	bArm2VertULD1Up_00 AT %MX26056.0 : BOOL;
	bArm2VertULD1Up_01 AT %MX26056.1 : BOOL;
	bArm2VertULD1Up_02 AT %MX26056.2 : BOOL;
	bArm2VertULD1Up_03 AT %MX26056.3 : BOOL;
	bArm2VertULD1Up_04 AT %MX26056.4 : BOOL;
	bArm2VertULD1Up_05 AT %MX26056.5 : BOOL;
	bArm2VertULD1Up_06 AT %MX26056.6 : BOOL;
	bArm2VertULD1Up_07 AT %MX26056.7 : BOOL;
	bArm2VertULD1Up_08 AT %MX26056.8 : BOOL;
	bArm2VertULD1Up_09 AT %MX26056.9 : BOOL;
	bArm2VertULD1Up_10 AT %MX26056.10 : BOOL;
	bArm2VertULD1Up_11 AT %MX26056.11 : BOOL;
	bArm2VertULD1Up_12 AT %MX26056.12 : BOOL;
	bArm2VertULD1Up_13 AT %MX26056.13 : BOOL;
	bArm2VertULD1Up_14 AT %MX26056.14 : BOOL;
	bArm2VertULD1Up_15 AT %MX26056.15 : BOOL;
	bArm2VertULD1Up_16 AT %MX26056.16 : BOOL;
	bArm2VertULD1Up_17 AT %MX26056.17 : BOOL;
	bArm2VertULD1Up_18 AT %MX26056.18 : BOOL;
	bArm2VertULD1Up_19 AT %MX26056.19 : BOOL;
	bArm2VertULD1Up_20 AT %MX26056.20 : BOOL;
	bArm2VertULD1Up_21 AT %MX26056.21 : BOOL;
	bArm2VertULD1Up_22 AT %MX26056.22 : BOOL;
	bArm2VertULD1Up_23 AT %MX26056.23 : BOOL;
	bArm2VertULD1Up_24 AT %MX26056.24 : BOOL;
	bArm2VertULD1Up_25 AT %MX26056.25 : BOOL;
	bArm2VertULD1Up_26 AT %MX26056.26 : BOOL;
	bArm2VertULD1Up_27 AT %MX26056.27 : BOOL;
	bArm2VertULD1Up_28 AT %MX26056.28 : BOOL;
	bArm2VertULD1Up_29 AT %MX26056.29 : BOOL;
	bArm2VertULD1Up_30 AT %MX26056.30 : BOOL;
	bArm2VertULD1Up_31 AT %MX26056.31 : BOOL;

	bArm2VertStn1Up_00 AT %MX26004.0 : BOOL;
	bArm2VertStn1Up_01 AT %MX26004.1 : BOOL;
	bArm2VertStn1Up_02 AT %MX26004.2 : BOOL;
	bArm2VertStn1Up_03 AT %MX26004.3 : BOOL;
	bArm2VertStn1Up_04 AT %MX26004.4 : BOOL;
	bArm2VertStn1Up_05 AT %MX26004.5 : BOOL;
	bArm2VertStn1Up_06 AT %MX26004.6 : BOOL;
	bArm2VertStn1Up_07 AT %MX26004.7 : BOOL;
	bArm2VertStn1Up_08 AT %MX26004.8 : BOOL;
	bArm2VertStn1Up_09 AT %MX26004.9 : BOOL;
	bArm2VertStn1Up_10 AT %MX26004.10 : BOOL;
	bArm2VertStn1Up_11 AT %MX26004.11 : BOOL;
	bArm2VertStn1Up_12 AT %MX26004.12 : BOOL;
	bArm2VertStn1Up_13 AT %MX26004.13 : BOOL;
	bArm2VertStn1Up_14 AT %MX26004.14 : BOOL;
	bArm2VertStn1Up_15 AT %MX26004.15 : BOOL;
	bArm2VertStn1Up_16 AT %MX26004.16 : BOOL;
	bArm2VertStn1Up_17 AT %MX26004.17 : BOOL;
	bArm2VertStn1Up_18 AT %MX26004.18 : BOOL;
	bArm2VertStn1Up_19 AT %MX26004.19 : BOOL;
	bArm2VertStn1Up_20 AT %MX26004.20 : BOOL;
	bArm2VertStn1Up_21 AT %MX26004.21 : BOOL;
	bArm2VertStn1Up_22 AT %MX26004.22 : BOOL;
	bArm2VertStn1Up_23 AT %MX26004.23 : BOOL;
	bArm2VertStn1Up_24 AT %MX26004.24 : BOOL;
	bArm2VertStn1Up_25 AT %MX26004.25 : BOOL;
	bArm2VertStn1Up_26 AT %MX26004.26 : BOOL;
	bArm2VertStn1Up_27 AT %MX26004.27 : BOOL;
	bArm2VertStn1Up_28 AT %MX26004.28 : BOOL;
	bArm2VertStn1Up_29 AT %MX26004.29 : BOOL;
	bArm2VertStn1Up_30 AT %MX26004.30 : BOOL;
	bArm2VertStn1Up_31 AT %MX26004.31 : BOOL;

	bArm2VertStn2Up_00 AT %MX26008.0 : BOOL;
	bArm2VertStn2Up_01 AT %MX26008.1 : BOOL;
	bArm2VertStn2Up_02 AT %MX26008.2 : BOOL;
	bArm2VertStn2Up_03 AT %MX26008.3 : BOOL;
	bArm2VertStn2Up_04 AT %MX26008.4 : BOOL;
	bArm2VertStn2Up_05 AT %MX26008.5 : BOOL;
	bArm2VertStn2Up_06 AT %MX26008.6 : BOOL;
	bArm2VertStn2Up_07 AT %MX26008.7 : BOOL;
	bArm2VertStn2Up_08 AT %MX26008.8 : BOOL;
	bArm2VertStn2Up_09 AT %MX26008.9 : BOOL;
	bArm2VertStn2Up_10 AT %MX26008.10 : BOOL;
	bArm2VertStn2Up_11 AT %MX26008.11 : BOOL;
	bArm2VertStn2Up_12 AT %MX26008.12 : BOOL;
	bArm2VertStn2Up_13 AT %MX26008.13 : BOOL;
	bArm2VertStn2Up_14 AT %MX26008.14 : BOOL;
	bArm2VertStn2Up_15 AT %MX26008.15 : BOOL;
	bArm2VertStn2Up_16 AT %MX26008.16 : BOOL;
	bArm2VertStn2Up_17 AT %MX26008.17 : BOOL;
	bArm2VertStn2Up_18 AT %MX26008.18 : BOOL;
	bArm2VertStn2Up_19 AT %MX26008.19 : BOOL;
	bArm2VertStn2Up_20 AT %MX26008.20 : BOOL;
	bArm2VertStn2Up_21 AT %MX26008.21 : BOOL;
	bArm2VertStn2Up_22 AT %MX26008.22 : BOOL;
	bArm2VertStn2Up_23 AT %MX26008.23 : BOOL;
	bArm2VertStn2Up_24 AT %MX26008.24 : BOOL;
	bArm2VertStn2Up_25 AT %MX26008.25 : BOOL;
	bArm2VertStn2Up_26 AT %MX26008.26 : BOOL;
	bArm2VertStn2Up_27 AT %MX26008.27 : BOOL;
	bArm2VertStn2Up_28 AT %MX26008.28 : BOOL;
	bArm2VertStn2Up_29 AT %MX26008.29 : BOOL;
	bArm2VertStn2Up_30 AT %MX26008.30 : BOOL;
	bArm2VertStn2Up_31 AT %MX26008.31 : BOOL;

	bArm2VertStn3Up_00 AT %MX26012.0 : BOOL;
	bArm2VertStn3Up_01 AT %MX26012.1 : BOOL;
	bArm2VertStn3Up_02 AT %MX26012.2 : BOOL;
	bArm2VertStn3Up_03 AT %MX26012.3 : BOOL;
	bArm2VertStn3Up_04 AT %MX26012.4 : BOOL;
	bArm2VertStn3Up_05 AT %MX26012.5 : BOOL;
	bArm2VertStn3Up_06 AT %MX26012.6 : BOOL;
	bArm2VertStn3Up_07 AT %MX26012.7 : BOOL;
	bArm2VertStn3Up_08 AT %MX26012.8 : BOOL;
	bArm2VertStn3Up_09 AT %MX26012.9 : BOOL;
	bArm2VertStn3Up_10 AT %MX26012.10 : BOOL;
	bArm2VertStn3Up_11 AT %MX26012.11 : BOOL;
	bArm2VertStn3Up_12 AT %MX26012.12 : BOOL;
	bArm2VertStn3Up_13 AT %MX26012.13 : BOOL;
	bArm2VertStn3Up_14 AT %MX26012.14 : BOOL;
	bArm2VertStn3Up_15 AT %MX26012.15 : BOOL;
	bArm2VertStn3Up_16 AT %MX26012.16 : BOOL;
	bArm2VertStn3Up_17 AT %MX26012.17 : BOOL;
	bArm2VertStn3Up_18 AT %MX26012.18 : BOOL;
	bArm2VertStn3Up_19 AT %MX26012.19 : BOOL;
	bArm2VertStn3Up_20 AT %MX26012.20 : BOOL;
	bArm2VertStn3Up_21 AT %MX26012.21 : BOOL;
	bArm2VertStn3Up_22 AT %MX26012.22 : BOOL;
	bArm2VertStn3Up_23 AT %MX26012.23 : BOOL;
	bArm2VertStn3Up_24 AT %MX26012.24 : BOOL;
	bArm2VertStn3Up_25 AT %MX26012.25 : BOOL;
	bArm2VertStn3Up_26 AT %MX26012.26 : BOOL;
	bArm2VertStn3Up_27 AT %MX26012.27 : BOOL;
	bArm2VertStn3Up_28 AT %MX26012.28 : BOOL;
	bArm2VertStn3Up_29 AT %MX26012.29 : BOOL;
	bArm2VertStn3Up_30 AT %MX26012.30 : BOOL;
	bArm2VertStn3Up_31 AT %MX26012.31 : BOOL;

	bArm2VertStn4Up_00 AT %MX26016.0 : BOOL;
	bArm2VertStn4Up_01 AT %MX26016.1 : BOOL;
	bArm2VertStn4Up_02 AT %MX26016.2 : BOOL;
	bArm2VertStn4Up_03 AT %MX26016.3 : BOOL;
	bArm2VertStn4Up_04 AT %MX26016.4 : BOOL;
	bArm2VertStn4Up_05 AT %MX26016.5 : BOOL;
	bArm2VertStn4Up_06 AT %MX26016.6 : BOOL;
	bArm2VertStn4Up_07 AT %MX26016.7 : BOOL;
	bArm2VertStn4Up_08 AT %MX26016.8 : BOOL;
	bArm2VertStn4Up_09 AT %MX26016.9 : BOOL;
	bArm2VertStn4Up_10 AT %MX26016.10 : BOOL;
	bArm2VertStn4Up_11 AT %MX26016.11 : BOOL;
	bArm2VertStn4Up_12 AT %MX26016.12 : BOOL;
	bArm2VertStn4Up_13 AT %MX26016.13 : BOOL;
	bArm2VertStn4Up_14 AT %MX26016.14 : BOOL;
	bArm2VertStn4Up_15 AT %MX26016.15 : BOOL;
	bArm2VertStn4Up_16 AT %MX26016.16 : BOOL;
	bArm2VertStn4Up_17 AT %MX26016.17 : BOOL;
	bArm2VertStn4Up_18 AT %MX26016.18 : BOOL;
	bArm2VertStn4Up_19 AT %MX26016.19 : BOOL;
	bArm2VertStn4Up_20 AT %MX26016.20 : BOOL;
	bArm2VertStn4Up_21 AT %MX26016.21 : BOOL;
	bArm2VertStn4Up_22 AT %MX26016.22 : BOOL;
	bArm2VertStn4Up_23 AT %MX26016.23 : BOOL;
	bArm2VertStn4Up_24 AT %MX26016.24 : BOOL;
	bArm2VertStn4Up_25 AT %MX26016.25 : BOOL;
	bArm2VertStn4Up_26 AT %MX26016.26 : BOOL;
	bArm2VertStn4Up_27 AT %MX26016.27 : BOOL;
	bArm2VertStn4Up_28 AT %MX26016.28 : BOOL;
	bArm2VertStn4Up_29 AT %MX26016.29 : BOOL;
	bArm2VertStn4Up_30 AT %MX26016.30 : BOOL;
	bArm2VertStn4Up_31 AT %MX26016.31 : BOOL;

	bArm2VertStn5Up_00 AT %MX26020.0 : BOOL;
	bArm2VertStn5Up_01 AT %MX26020.1 : BOOL;
	bArm2VertStn5Up_02 AT %MX26020.2 : BOOL;
	bArm2VertStn5Up_03 AT %MX26020.3 : BOOL;
	bArm2VertStn5Up_04 AT %MX26020.4 : BOOL;
	bArm2VertStn5Up_05 AT %MX26020.5 : BOOL;
	bArm2VertStn5Up_06 AT %MX26020.6 : BOOL;
	bArm2VertStn5Up_07 AT %MX26020.7 : BOOL;
	bArm2VertStn5Up_08 AT %MX26020.8 : BOOL;
	bArm2VertStn5Up_09 AT %MX26020.9 : BOOL;
	bArm2VertStn5Up_10 AT %MX26020.10 : BOOL;
	bArm2VertStn5Up_11 AT %MX26020.11 : BOOL;
	bArm2VertStn5Up_12 AT %MX26020.12 : BOOL;
	bArm2VertStn5Up_13 AT %MX26020.13 : BOOL;
	bArm2VertStn5Up_14 AT %MX26020.14 : BOOL;
	bArm2VertStn5Up_15 AT %MX26020.15 : BOOL;
	bArm2VertStn5Up_16 AT %MX26020.16 : BOOL;
	bArm2VertStn5Up_17 AT %MX26020.17 : BOOL;
	bArm2VertStn5Up_18 AT %MX26020.18 : BOOL;
	bArm2VertStn5Up_19 AT %MX26020.19 : BOOL;
	bArm2VertStn5Up_20 AT %MX26020.20 : BOOL;
	bArm2VertStn5Up_21 AT %MX26020.21 : BOOL;
	bArm2VertStn5Up_22 AT %MX26020.22 : BOOL;
	bArm2VertStn5Up_23 AT %MX26020.23 : BOOL;
	bArm2VertStn5Up_24 AT %MX26020.24 : BOOL;
	bArm2VertStn5Up_25 AT %MX26020.25 : BOOL;
	bArm2VertStn5Up_26 AT %MX26020.26 : BOOL;
	bArm2VertStn5Up_27 AT %MX26020.27 : BOOL;
	bArm2VertStn5Up_28 AT %MX26020.28 : BOOL;
	bArm2VertStn5Up_29 AT %MX26020.29 : BOOL;
	bArm2VertStn5Up_30 AT %MX26020.30 : BOOL;
	bArm2VertStn5Up_31 AT %MX26020.31 : BOOL;

	bArm2VertStn6Up_00 AT %MX26024.0 : BOOL;
	bArm2VertStn6Up_01 AT %MX26024.1 : BOOL;
	bArm2VertStn6Up_02 AT %MX26024.2 : BOOL;
	bArm2VertStn6Up_03 AT %MX26024.3 : BOOL;
	bArm2VertStn6Up_04 AT %MX26024.4 : BOOL;
	bArm2VertStn6Up_05 AT %MX26024.5 : BOOL;
	bArm2VertStn6Up_06 AT %MX26024.6 : BOOL;
	bArm2VertStn6Up_07 AT %MX26024.7 : BOOL;
	bArm2VertStn6Up_08 AT %MX26024.8 : BOOL;
	bArm2VertStn6Up_09 AT %MX26024.9 : BOOL;
	bArm2VertStn6Up_10 AT %MX26024.10 : BOOL;
	bArm2VertStn6Up_11 AT %MX26024.11 : BOOL;
	bArm2VertStn6Up_12 AT %MX26024.12 : BOOL;
	bArm2VertStn6Up_13 AT %MX26024.13 : BOOL;
	bArm2VertStn6Up_14 AT %MX26024.14 : BOOL;
	bArm2VertStn6Up_15 AT %MX26024.15 : BOOL;
	bArm2VertStn6Up_16 AT %MX26024.16 : BOOL;
	bArm2VertStn6Up_17 AT %MX26024.17 : BOOL;
	bArm2VertStn6Up_18 AT %MX26024.18 : BOOL;
	bArm2VertStn6Up_19 AT %MX26024.19 : BOOL;
	bArm2VertStn6Up_20 AT %MX26024.20 : BOOL;
	bArm2VertStn6Up_21 AT %MX26024.21 : BOOL;
	bArm2VertStn6Up_22 AT %MX26024.22 : BOOL;
	bArm2VertStn6Up_23 AT %MX26024.23 : BOOL;
	bArm2VertStn6Up_24 AT %MX26024.24 : BOOL;
	bArm2VertStn6Up_25 AT %MX26024.25 : BOOL;
	bArm2VertStn6Up_26 AT %MX26024.26 : BOOL;
	bArm2VertStn6Up_27 AT %MX26024.27 : BOOL;
	bArm2VertStn6Up_28 AT %MX26024.28 : BOOL;
	bArm2VertStn6Up_29 AT %MX26024.29 : BOOL;
	bArm2VertStn6Up_30 AT %MX26024.30 : BOOL;
	bArm2VertStn6Up_31 AT %MX26024.31 : BOOL;

	bArm2VertStn7Up_00 AT %MX26028.0 : BOOL;
	bArm2VertStn7Up_01 AT %MX26028.1 : BOOL;
	bArm2VertStn7Up_02 AT %MX26028.2 : BOOL;
	bArm2VertStn7Up_03 AT %MX26028.3 : BOOL;
	bArm2VertStn7Up_04 AT %MX26028.4 : BOOL;
	bArm2VertStn7Up_05 AT %MX26028.5 : BOOL;
	bArm2VertStn7Up_06 AT %MX26028.6 : BOOL;
	bArm2VertStn7Up_07 AT %MX26028.7 : BOOL;
	bArm2VertStn7Up_08 AT %MX26028.8 : BOOL;
	bArm2VertStn7Up_09 AT %MX26028.9 : BOOL;
	bArm2VertStn7Up_10 AT %MX26028.10 : BOOL;
	bArm2VertStn7Up_11 AT %MX26028.11 : BOOL;
	bArm2VertStn7Up_12 AT %MX26028.12 : BOOL;
	bArm2VertStn7Up_13 AT %MX26028.13 : BOOL;
	bArm2VertStn7Up_14 AT %MX26028.14 : BOOL;
	bArm2VertStn7Up_15 AT %MX26028.15 : BOOL;
	bArm2VertStn7Up_16 AT %MX26028.16 : BOOL;
	bArm2VertStn7Up_17 AT %MX26028.17 : BOOL;
	bArm2VertStn7Up_18 AT %MX26028.18 : BOOL;
	bArm2VertStn7Up_19 AT %MX26028.19 : BOOL;
	bArm2VertStn7Up_20 AT %MX26028.20 : BOOL;
	bArm2VertStn7Up_21 AT %MX26028.21 : BOOL;
	bArm2VertStn7Up_22 AT %MX26028.22 : BOOL;
	bArm2VertStn7Up_23 AT %MX26028.23 : BOOL;
	bArm2VertStn7Up_24 AT %MX26028.24 : BOOL;
	bArm2VertStn7Up_25 AT %MX26028.25 : BOOL;
	bArm2VertStn7Up_26 AT %MX26028.26 : BOOL;
	bArm2VertStn7Up_27 AT %MX26028.27 : BOOL;
	bArm2VertStn7Up_28 AT %MX26028.28 : BOOL;
	bArm2VertStn7Up_29 AT %MX26028.29 : BOOL;
	bArm2VertStn7Up_30 AT %MX26028.30 : BOOL;
	bArm2VertStn7Up_31 AT %MX26028.31 : BOOL;

	bArm2VertStn8Up_00 AT %MX26032.0 : BOOL;
	bArm2VertStn8Up_01 AT %MX26032.1 : BOOL;
	bArm2VertStn8Up_02 AT %MX26032.2 : BOOL;
	bArm2VertStn8Up_03 AT %MX26032.3 : BOOL;
	bArm2VertStn8Up_04 AT %MX26032.4 : BOOL;
	bArm2VertStn8Up_05 AT %MX26032.5 : BOOL;
	bArm2VertStn8Up_06 AT %MX26032.6 : BOOL;
	bArm2VertStn8Up_07 AT %MX26032.7 : BOOL;
	bArm2VertStn8Up_08 AT %MX26032.8 : BOOL;
	bArm2VertStn8Up_09 AT %MX26032.9 : BOOL;
	bArm2VertStn8Up_10 AT %MX26032.10 : BOOL;
	bArm2VertStn8Up_11 AT %MX26032.11 : BOOL;
	bArm2VertStn8Up_12 AT %MX26032.12 : BOOL;
	bArm2VertStn8Up_13 AT %MX26032.13 : BOOL;
	bArm2VertStn8Up_14 AT %MX26032.14 : BOOL;
	bArm2VertStn8Up_15 AT %MX26032.15 : BOOL;
	bArm2VertStn8Up_16 AT %MX26032.16 : BOOL;
	bArm2VertStn8Up_17 AT %MX26032.17 : BOOL;
	bArm2VertStn8Up_18 AT %MX26032.18 : BOOL;
	bArm2VertStn8Up_19 AT %MX26032.19 : BOOL;
	bArm2VertStn8Up_20 AT %MX26032.20 : BOOL;
	bArm2VertStn8Up_21 AT %MX26032.21 : BOOL;
	bArm2VertStn8Up_22 AT %MX26032.22 : BOOL;
	bArm2VertStn8Up_23 AT %MX26032.23 : BOOL;
	bArm2VertStn8Up_24 AT %MX26032.24 : BOOL;
	bArm2VertStn8Up_25 AT %MX26032.25 : BOOL;
	bArm2VertStn8Up_26 AT %MX26032.26 : BOOL;
	bArm2VertStn8Up_27 AT %MX26032.27 : BOOL;
	bArm2VertStn8Up_28 AT %MX26032.28 : BOOL;
	bArm2VertStn8Up_29 AT %MX26032.29 : BOOL;
	bArm2VertStn8Up_30 AT %MX26032.30 : BOOL;
	bArm2VertStn8Up_31 AT %MX26032.31 : BOOL;

	bArm2VertStn9Up_00 AT %MX26036.0 : BOOL;
	bArm2VertStn9Up_01 AT %MX26036.1 : BOOL;
	bArm2VertStn9Up_02 AT %MX26036.2 : BOOL;
	bArm2VertStn9Up_03 AT %MX26036.3 : BOOL;
	bArm2VertStn9Up_04 AT %MX26036.4 : BOOL;
	bArm2VertStn9Up_05 AT %MX26036.5 : BOOL;
	bArm2VertStn9Up_06 AT %MX26036.6 : BOOL;
	bArm2VertStn9Up_07 AT %MX26036.7 : BOOL;
	bArm2VertStn9Up_08 AT %MX26036.8 : BOOL;
	bArm2VertStn9Up_09 AT %MX26036.9 : BOOL;
	bArm2VertStn9Up_10 AT %MX26036.10 : BOOL;
	bArm2VertStn9Up_11 AT %MX26036.11 : BOOL;
	bArm2VertStn9Up_12 AT %MX26036.12 : BOOL;
	bArm2VertStn9Up_13 AT %MX26036.13 : BOOL;
	bArm2VertStn9Up_14 AT %MX26036.14 : BOOL;
	bArm2VertStn9Up_15 AT %MX26036.15 : BOOL;
	bArm2VertStn9Up_16 AT %MX26036.16 : BOOL;
	bArm2VertStn9Up_17 AT %MX26036.17 : BOOL;
	bArm2VertStn9Up_18 AT %MX26036.18 : BOOL;
	bArm2VertStn9Up_19 AT %MX26036.19 : BOOL;
	bArm2VertStn9Up_20 AT %MX26036.20 : BOOL;
	bArm2VertStn9Up_21 AT %MX26036.21 : BOOL;
	bArm2VertStn9Up_22 AT %MX26036.22 : BOOL;
	bArm2VertStn9Up_23 AT %MX26036.23 : BOOL;
	bArm2VertStn9Up_24 AT %MX26036.24 : BOOL;
	bArm2VertStn9Up_25 AT %MX26036.25 : BOOL;
	bArm2VertStn9Up_26 AT %MX26036.26 : BOOL;
	bArm2VertStn9Up_27 AT %MX26036.27 : BOOL;
	bArm2VertStn9Up_28 AT %MX26036.28 : BOOL;
	bArm2VertStn9Up_29 AT %MX26036.29 : BOOL;
	bArm2VertStn9Up_30 AT %MX26036.30 : BOOL;
	bArm2VertStn9Up_31 AT %MX26036.31 : BOOL;

	bArm2VertStn10Up_00 AT %MX26040.0 : BOOL;
	bArm2VertStn10Up_01 AT %MX26040.1 : BOOL;
	bArm2VertStn10Up_02 AT %MX26040.2 : BOOL;
	bArm2VertStn10Up_03 AT %MX26040.3 : BOOL;
	bArm2VertStn10Up_04 AT %MX26040.4 : BOOL;
	bArm2VertStn10Up_05 AT %MX26040.5 : BOOL;
	bArm2VertStn10Up_06 AT %MX26040.6 : BOOL;
	bArm2VertStn10Up_07 AT %MX26040.7 : BOOL;
	bArm2VertStn10Up_08 AT %MX26040.8 : BOOL;
	bArm2VertStn10Up_09 AT %MX26040.9 : BOOL;
	bArm2VertStn10Up_10 AT %MX26040.10 : BOOL;
	bArm2VertStn10Up_11 AT %MX26040.11 : BOOL;
	bArm2VertStn10Up_12 AT %MX26040.12 : BOOL;
	bArm2VertStn10Up_13 AT %MX26040.13 : BOOL;
	bArm2VertStn10Up_14 AT %MX26040.14 : BOOL;
	bArm2VertStn10Up_15 AT %MX26040.15 : BOOL;
	bArm2VertStn10Up_16 AT %MX26040.16 : BOOL;
	bArm2VertStn10Up_17 AT %MX26040.17 : BOOL;
	bArm2VertStn10Up_18 AT %MX26040.18 : BOOL;
	bArm2VertStn10Up_19 AT %MX26040.19 : BOOL;
	bArm2VertStn10Up_20 AT %MX26040.20 : BOOL;
	bArm2VertStn10Up_21 AT %MX26040.21 : BOOL;
	bArm2VertStn10Up_22 AT %MX26040.22 : BOOL;
	bArm2VertStn10Up_23 AT %MX26040.23 : BOOL;
	bArm2VertStn10Up_24 AT %MX26040.24 : BOOL;
	bArm2VertStn10Up_25 AT %MX26040.25 : BOOL;
	bArm2VertStn10Up_26 AT %MX26040.26 : BOOL;
	bArm2VertStn10Up_27 AT %MX26040.27 : BOOL;
	bArm2VertStn10Up_28 AT %MX26040.28 : BOOL;
	bArm2VertStn10Up_29 AT %MX26040.29 : BOOL;
	bArm2VertStn10Up_30 AT %MX26040.30 : BOOL;
	bArm2VertStn10Up_31 AT %MX26040.31 : BOOL;

	bArm2VertStn11Up_00 AT %MX26044.0 : BOOL;
	bArm2VertStn11Up_01 AT %MX26044.1 : BOOL;
	bArm2VertStn11Up_02 AT %MX26044.2 : BOOL;
	bArm2VertStn11Up_03 AT %MX26044.3 : BOOL;
	bArm2VertStn11Up_04 AT %MX26044.4 : BOOL;
	bArm2VertStn11Up_05 AT %MX26044.5 : BOOL;
	bArm2VertStn11Up_06 AT %MX26044.6 : BOOL;
	bArm2VertStn11Up_07 AT %MX26044.7 : BOOL;
	bArm2VertStn11Up_08 AT %MX26044.8 : BOOL;
	bArm2VertStn11Up_09 AT %MX26044.9 : BOOL;
	bArm2VertStn11Up_10 AT %MX26044.10 : BOOL;
	bArm2VertStn11Up_11 AT %MX26044.11 : BOOL;
	bArm2VertStn11Up_12 AT %MX26044.12 : BOOL;
	bArm2VertStn11Up_13 AT %MX26044.13 : BOOL;
	bArm2VertStn11Up_14 AT %MX26044.14 : BOOL;
	bArm2VertStn11Up_15 AT %MX26044.15 : BOOL;
	bArm2VertStn11Up_16 AT %MX26044.16 : BOOL;
	bArm2VertStn11Up_17 AT %MX26044.17 : BOOL;
	bArm2VertStn11Up_18 AT %MX26044.18 : BOOL;
	bArm2VertStn11Up_19 AT %MX26044.19 : BOOL;
	bArm2VertStn11Up_20 AT %MX26044.20 : BOOL;
	bArm2VertStn11Up_21 AT %MX26044.21 : BOOL;
	bArm2VertStn11Up_22 AT %MX26044.22 : BOOL;
	bArm2VertStn11Up_23 AT %MX26044.23 : BOOL;
	bArm2VertStn11Up_24 AT %MX26044.24 : BOOL;
	bArm2VertStn11Up_25 AT %MX26044.25 : BOOL;
	bArm2VertStn11Up_26 AT %MX26044.26 : BOOL;
	bArm2VertStn11Up_27 AT %MX26044.27 : BOOL;
	bArm2VertStn11Up_28 AT %MX26044.28 : BOOL;
	bArm2VertStn11Up_29 AT %MX26044.29 : BOOL;
	bArm2VertStn11Up_30 AT %MX26044.30 : BOOL;
	bArm2VertStn11Up_31 AT %MX26044.31 : BOOL;

	bArm2VertStn12Up_00 AT %MX26048.0 : BOOL;
	bArm2VertStn12Up_01 AT %MX26048.1 : BOOL;
	bArm2VertStn12Up_02 AT %MX26048.2 : BOOL;
	bArm2VertStn12Up_03 AT %MX26048.3 : BOOL;
	bArm2VertStn12Up_04 AT %MX26048.4 : BOOL;
	bArm2VertStn12Up_05 AT %MX26048.5 : BOOL;
	bArm2VertStn12Up_06 AT %MX26048.6 : BOOL;
	bArm2VertStn12Up_07 AT %MX26048.7 : BOOL;
	bArm2VertStn12Up_08 AT %MX26048.8 : BOOL;
	bArm2VertStn12Up_09 AT %MX26048.9 : BOOL;
	bArm2VertStn12Up_10 AT %MX26048.10 : BOOL;
	bArm2VertStn12Up_11 AT %MX26048.11 : BOOL;
	bArm2VertStn12Up_12 AT %MX26048.12 : BOOL;
	bArm2VertStn12Up_13 AT %MX26048.13 : BOOL;
	bArm2VertStn12Up_14 AT %MX26048.14 : BOOL;
	bArm2VertStn12Up_15 AT %MX26048.15 : BOOL;
	bArm2VertStn12Up_16 AT %MX26048.16 : BOOL;
	bArm2VertStn12Up_17 AT %MX26048.17 : BOOL;
	bArm2VertStn12Up_18 AT %MX26048.18 : BOOL;
	bArm2VertStn12Up_19 AT %MX26048.19 : BOOL;
	bArm2VertStn12Up_20 AT %MX26048.20 : BOOL;
	bArm2VertStn12Up_21 AT %MX26048.21 : BOOL;
	bArm2VertStn12Up_22 AT %MX26048.22 : BOOL;
	bArm2VertStn12Up_23 AT %MX26048.23 : BOOL;
	bArm2VertStn12Up_24 AT %MX26048.24 : BOOL;
	bArm2VertStn12Up_25 AT %MX26048.25 : BOOL;
	bArm2VertStn12Up_26 AT %MX26048.26 : BOOL;
	bArm2VertStn12Up_27 AT %MX26048.27 : BOOL;
	bArm2VertStn12Up_28 AT %MX26048.28 : BOOL;
	bArm2VertStn12Up_29 AT %MX26048.29 : BOOL;
	bArm2VertStn12Up_30 AT %MX26048.30 : BOOL;
	bArm2VertStn12Up_31 AT %MX26048.31 : BOOL;

(* xxxxxxxxxxxxxxxxxxxxxxxxxxxxxxxxxxxxxxx Vert xxxxxxxxxxxxxxxxxxxxxxxxxxxxxxxxxxxxxxx*)
(*========= Down SpSlanted BOOL LINK with %MX26100-MX26199 =========*)

	bArm2VertStn1SpSlanted_00 AT %MX26104.0 : BOOL;
	bArm2VertStn1SpSlanted_01 AT %MX26104.1 : BOOL;
	bArm2VertStn1SpSlanted_02 AT %MX26104.2 : BOOL;
	bArm2VertStn1SpSlanted_03 AT %MX26104.3 : BOOL;
	bArm2VertStn1SpSlanted_04 AT %MX26104.4 : BOOL;
	bArm2VertStn1SpSlanted_05 AT %MX26104.5 : BOOL;
	bArm2VertStn1SpSlanted_06 AT %MX26104.6 : BOOL;
	bArm2VertStn1SpSlanted_07 AT %MX26104.7 : BOOL;
	bArm2VertStn1SpSlanted_08 AT %MX26104.8 : BOOL;
	bArm2VertStn1SpSlanted_09 AT %MX26104.9 : BOOL;
	bArm2VertStn1SpSlanted_10 AT %MX26104.10 : BOOL;
	bArm2VertStn1SpSlanted_11 AT %MX26104.11 : BOOL;
	bArm2VertStn1SpSlanted_12 AT %MX26104.12 : BOOL;
	bArm2VertStn1SpSlanted_13 AT %MX26104.13 : BOOL;
	bArm2VertStn1SpSlanted_14 AT %MX26104.14 : BOOL;
	bArm2VertStn1SpSlanted_15 AT %MX26104.15 : BOOL;
	bArm2VertStn1SpSlanted_16 AT %MX26104.16 : BOOL;
	bArm2VertStn1SpSlanted_17 AT %MX26104.17 : BOOL;
	bArm2VertStn1SpSlanted_18 AT %MX26104.18 : BOOL;
	bArm2VertStn1SpSlanted_19 AT %MX26104.19 : BOOL;
	bArm2VertStn1SpSlanted_20 AT %MX26104.20 : BOOL;
	bArm2VertStn1SpSlanted_21 AT %MX26104.21 : BOOL;
	bArm2VertStn1SpSlanted_22 AT %MX26104.22 : BOOL;
	bArm2VertStn1SpSlanted_23 AT %MX26104.23 : BOOL;
	bArm2VertStn1SpSlanted_24 AT %MX26104.24 : BOOL;
	bArm2VertStn1SpSlanted_25 AT %MX26104.25 : BOOL;
	bArm2VertStn1SpSlanted_26 AT %MX26104.26 : BOOL;
	bArm2VertStn1SpSlanted_27 AT %MX26104.27 : BOOL;
	bArm2VertStn1SpSlanted_28 AT %MX26104.28 : BOOL;
	bArm2VertStn1SpSlanted_29 AT %MX26104.29 : BOOL;
	bArm2VertStn1SpSlanted_30 AT %MX26104.30 : BOOL;
	bArm2VertStn1SpSlanted_31 AT %MX26104.31 : BOOL;

	bArm2VertStn2SpSlanted_00 AT %MX26108.0 : BOOL;
	bArm2VertStn2SpSlanted_01 AT %MX26108.1 : BOOL;
	bArm2VertStn2SpSlanted_02 AT %MX26108.2 : BOOL;
	bArm2VertStn2SpSlanted_03 AT %MX26108.3 : BOOL;
	bArm2VertStn2SpSlanted_04 AT %MX26108.4 : BOOL;
	bArm2VertStn2SpSlanted_05 AT %MX26108.5 : BOOL;
	bArm2VertStn2SpSlanted_06 AT %MX26108.6 : BOOL;
	bArm2VertStn2SpSlanted_07 AT %MX26108.7 : BOOL;
	bArm2VertStn2SpSlanted_08 AT %MX26108.8 : BOOL;
	bArm2VertStn2SpSlanted_09 AT %MX26108.9 : BOOL;
	bArm2VertStn2SpSlanted_10 AT %MX26108.10 : BOOL;
	bArm2VertStn2SpSlanted_11 AT %MX26108.11 : BOOL;
	bArm2VertStn2SpSlanted_12 AT %MX26108.12 : BOOL;
	bArm2VertStn2SpSlanted_13 AT %MX26108.13 : BOOL;
	bArm2VertStn2SpSlanted_14 AT %MX26108.14 : BOOL;
	bArm2VertStn2SpSlanted_15 AT %MX26108.15 : BOOL;
	bArm2VertStn2SpSlanted_16 AT %MX26108.16 : BOOL;
	bArm2VertStn2SpSlanted_17 AT %MX26108.17 : BOOL;
	bArm2VertStn2SpSlanted_18 AT %MX26108.18 : BOOL;
	bArm2VertStn2SpSlanted_19 AT %MX26108.19 : BOOL;
	bArm2VertStn2SpSlanted_20 AT %MX26108.20 : BOOL;
	bArm2VertStn2SpSlanted_21 AT %MX26108.21 : BOOL;
	bArm2VertStn2SpSlanted_22 AT %MX26108.22 : BOOL;
	bArm2VertStn2SpSlanted_23 AT %MX26108.23 : BOOL;
	bArm2VertStn2SpSlanted_24 AT %MX26108.24 : BOOL;
	bArm2VertStn2SpSlanted_25 AT %MX26108.25 : BOOL;
	bArm2VertStn2SpSlanted_26 AT %MX26108.26 : BOOL;
	bArm2VertStn2SpSlanted_27 AT %MX26108.27 : BOOL;
	bArm2VertStn2SpSlanted_28 AT %MX26108.28 : BOOL;
	bArm2VertStn2SpSlanted_29 AT %MX26108.29 : BOOL;
	bArm2VertStn2SpSlanted_30 AT %MX26108.30 : BOOL;
	bArm2VertStn2SpSlanted_31 AT %MX26108.31 : BOOL;

	bArm2VertStn3SpSlanted_00 AT %MX26112.0 : BOOL;
	bArm2VertStn3SpSlanted_01 AT %MX26112.1 : BOOL;
	bArm2VertStn3SpSlanted_02 AT %MX26112.2 : BOOL;
	bArm2VertStn3SpSlanted_03 AT %MX26112.3 : BOOL;
	bArm2VertStn3SpSlanted_04 AT %MX26112.4 : BOOL;
	bArm2VertStn3SpSlanted_05 AT %MX26112.5 : BOOL;
	bArm2VertStn3SpSlanted_06 AT %MX26112.6 : BOOL;
	bArm2VertStn3SpSlanted_07 AT %MX26112.7 : BOOL;
	bArm2VertStn3SpSlanted_08 AT %MX26112.8 : BOOL;
	bArm2VertStn3SpSlanted_09 AT %MX26112.9 : BOOL;
	bArm2VertStn3SpSlanted_10 AT %MX26112.10 : BOOL;
	bArm2VertStn3SpSlanted_11 AT %MX26112.11 : BOOL;
	bArm2VertStn3SpSlanted_12 AT %MX26112.12 : BOOL;
	bArm2VertStn3SpSlanted_13 AT %MX26112.13 : BOOL;
	bArm2VertStn3SpSlanted_14 AT %MX26112.14 : BOOL;
	bArm2VertStn3SpSlanted_15 AT %MX26112.15 : BOOL;
	bArm2VertStn3SpSlanted_16 AT %MX26112.16 : BOOL;
	bArm2VertStn3SpSlanted_17 AT %MX26112.17 : BOOL;
	bArm2VertStn3SpSlanted_18 AT %MX26112.18 : BOOL;
	bArm2VertStn3SpSlanted_19 AT %MX26112.19 : BOOL;
	bArm2VertStn3SpSlanted_20 AT %MX26112.20 : BOOL;
	bArm2VertStn3SpSlanted_21 AT %MX26112.21 : BOOL;
	bArm2VertStn3SpSlanted_22 AT %MX26112.22 : BOOL;
	bArm2VertStn3SpSlanted_23 AT %MX26112.23 : BOOL;
	bArm2VertStn3SpSlanted_24 AT %MX26112.24 : BOOL;
	bArm2VertStn3SpSlanted_25 AT %MX26112.25 : BOOL;
	bArm2VertStn3SpSlanted_26 AT %MX26112.26 : BOOL;
	bArm2VertStn3SpSlanted_27 AT %MX26112.27 : BOOL;
	bArm2VertStn3SpSlanted_28 AT %MX26112.28 : BOOL;
	bArm2VertStn3SpSlanted_29 AT %MX26112.29 : BOOL;
	bArm2VertStn3SpSlanted_30 AT %MX26112.30 : BOOL;
	bArm2VertStn3SpSlanted_31 AT %MX26112.31 : BOOL;

	bArm2VertStn4SpSlanted_00 AT %MX26116.0 : BOOL;
	bArm2VertStn4SpSlanted_01 AT %MX26116.1 : BOOL;
	bArm2VertStn4SpSlanted_02 AT %MX26116.2 : BOOL;
	bArm2VertStn4SpSlanted_03 AT %MX26116.3 : BOOL;
	bArm2VertStn4SpSlanted_04 AT %MX26116.4 : BOOL;
	bArm2VertStn4SpSlanted_05 AT %MX26116.5 : BOOL;
	bArm2VertStn4SpSlanted_06 AT %MX26116.6 : BOOL;
	bArm2VertStn4SpSlanted_07 AT %MX26116.7 : BOOL;
	bArm2VertStn4SpSlanted_08 AT %MX26116.8 : BOOL;
	bArm2VertStn4SpSlanted_09 AT %MX26116.9 : BOOL;
	bArm2VertStn4SpSlanted_10 AT %MX26116.10 : BOOL;
	bArm2VertStn4SpSlanted_11 AT %MX26116.11 : BOOL;
	bArm2VertStn4SpSlanted_12 AT %MX26116.12 : BOOL;
	bArm2VertStn4SpSlanted_13 AT %MX26116.13 : BOOL;
	bArm2VertStn4SpSlanted_14 AT %MX26116.14 : BOOL;
	bArm2VertStn4SpSlanted_15 AT %MX26116.15 : BOOL;
	bArm2VertStn4SpSlanted_16 AT %MX26116.16 : BOOL;
	bArm2VertStn4SpSlanted_17 AT %MX26116.17 : BOOL;
	bArm2VertStn4SpSlanted_18 AT %MX26116.18 : BOOL;
	bArm2VertStn4SpSlanted_19 AT %MX26116.19 : BOOL;
	bArm2VertStn4SpSlanted_20 AT %MX26116.20 : BOOL;
	bArm2VertStn4SpSlanted_21 AT %MX26116.21 : BOOL;
	bArm2VertStn4SpSlanted_22 AT %MX26116.22 : BOOL;
	bArm2VertStn4SpSlanted_23 AT %MX26116.23 : BOOL;
	bArm2VertStn4SpSlanted_24 AT %MX26116.24 : BOOL;
	bArm2VertStn4SpSlanted_25 AT %MX26116.25 : BOOL;
	bArm2VertStn4SpSlanted_26 AT %MX26116.26 : BOOL;
	bArm2VertStn4SpSlanted_27 AT %MX26116.27 : BOOL;
	bArm2VertStn4SpSlanted_28 AT %MX26116.28 : BOOL;
	bArm2VertStn4SpSlanted_29 AT %MX26116.29 : BOOL;
	bArm2VertStn4SpSlanted_30 AT %MX26116.30 : BOOL;
	bArm2VertStn4SpSlanted_31 AT %MX26116.31 : BOOL;

	bArm2VertStn5SpSlanted_00 AT %MX26120.0 : BOOL;
	bArm2VertStn5SpSlanted_01 AT %MX26120.1 : BOOL;
	bArm2VertStn5SpSlanted_02 AT %MX26120.2 : BOOL;
	bArm2VertStn5SpSlanted_03 AT %MX26120.3 : BOOL;
	bArm2VertStn5SpSlanted_04 AT %MX26120.4 : BOOL;
	bArm2VertStn5SpSlanted_05 AT %MX26120.5 : BOOL;
	bArm2VertStn5SpSlanted_06 AT %MX26120.6 : BOOL;
	bArm2VertStn5SpSlanted_07 AT %MX26120.7 : BOOL;
	bArm2VertStn5SpSlanted_08 AT %MX26120.8 : BOOL;
	bArm2VertStn5SpSlanted_09 AT %MX26120.9 : BOOL;
	bArm2VertStn5SpSlanted_10 AT %MX26120.10 : BOOL;
	bArm2VertStn5SpSlanted_11 AT %MX26120.11 : BOOL;
	bArm2VertStn5SpSlanted_12 AT %MX26120.12 : BOOL;
	bArm2VertStn5SpSlanted_13 AT %MX26120.13 : BOOL;
	bArm2VertStn5SpSlanted_14 AT %MX26120.14 : BOOL;
	bArm2VertStn5SpSlanted_15 AT %MX26120.15 : BOOL;
	bArm2VertStn5SpSlanted_16 AT %MX26120.16 : BOOL;
	bArm2VertStn5SpSlanted_17 AT %MX26120.17 : BOOL;
	bArm2VertStn5SpSlanted_18 AT %MX26120.18 : BOOL;
	bArm2VertStn5SpSlanted_19 AT %MX26120.19 : BOOL;
	bArm2VertStn5SpSlanted_20 AT %MX26120.20 : BOOL;
	bArm2VertStn5SpSlanted_21 AT %MX26120.21 : BOOL;
	bArm2VertStn5SpSlanted_22 AT %MX26120.22 : BOOL;
	bArm2VertStn5SpSlanted_23 AT %MX26120.23 : BOOL;
	bArm2VertStn5SpSlanted_24 AT %MX26120.24 : BOOL;
	bArm2VertStn5SpSlanted_25 AT %MX26120.25 : BOOL;
	bArm2VertStn5SpSlanted_26 AT %MX26120.26 : BOOL;
	bArm2VertStn5SpSlanted_27 AT %MX26120.27 : BOOL;
	bArm2VertStn5SpSlanted_28 AT %MX26120.28 : BOOL;
	bArm2VertStn5SpSlanted_29 AT %MX26120.29 : BOOL;
	bArm2VertStn5SpSlanted_30 AT %MX26120.30 : BOOL;
	bArm2VertStn5SpSlanted_31 AT %MX26120.31 : BOOL;

	bArm2VertStn6SpSlanted_00 AT %MX26124.0 : BOOL;
	bArm2VertStn6SpSlanted_01 AT %MX26124.1 : BOOL;
	bArm2VertStn6SpSlanted_02 AT %MX26124.2 : BOOL;
	bArm2VertStn6SpSlanted_03 AT %MX26124.3 : BOOL;
	bArm2VertStn6SpSlanted_04 AT %MX26124.4 : BOOL;
	bArm2VertStn6SpSlanted_05 AT %MX26124.5 : BOOL;
	bArm2VertStn6SpSlanted_06 AT %MX26124.6 : BOOL;
	bArm2VertStn6SpSlanted_07 AT %MX26124.7 : BOOL;
	bArm2VertStn6SpSlanted_08 AT %MX26124.8 : BOOL;
	bArm2VertStn6SpSlanted_09 AT %MX26124.9 : BOOL;
	bArm2VertStn6SpSlanted_10 AT %MX26124.10 : BOOL;
	bArm2VertStn6SpSlanted_11 AT %MX26124.11 : BOOL;
	bArm2VertStn6SpSlanted_12 AT %MX26124.12 : BOOL;
	bArm2VertStn6SpSlanted_13 AT %MX26124.13 : BOOL;
	bArm2VertStn6SpSlanted_14 AT %MX26124.14 : BOOL;
	bArm2VertStn6SpSlanted_15 AT %MX26124.15 : BOOL;
	bArm2VertStn6SpSlanted_16 AT %MX26124.16 : BOOL;
	bArm2VertStn6SpSlanted_17 AT %MX26124.17 : BOOL;
	bArm2VertStn6SpSlanted_18 AT %MX26124.18 : BOOL;
	bArm2VertStn6SpSlanted_19 AT %MX26124.19 : BOOL;
	bArm2VertStn6SpSlanted_20 AT %MX26124.20 : BOOL;
	bArm2VertStn6SpSlanted_21 AT %MX26124.21 : BOOL;
	bArm2VertStn6SpSlanted_22 AT %MX26124.22 : BOOL;
	bArm2VertStn6SpSlanted_23 AT %MX26124.23 : BOOL;
	bArm2VertStn6SpSlanted_24 AT %MX26124.24 : BOOL;
	bArm2VertStn6SpSlanted_25 AT %MX26124.25 : BOOL;
	bArm2VertStn6SpSlanted_26 AT %MX26124.26 : BOOL;
	bArm2VertStn6SpSlanted_27 AT %MX26124.27 : BOOL;
	bArm2VertStn6SpSlanted_28 AT %MX26124.28 : BOOL;
	bArm2VertStn6SpSlanted_29 AT %MX26124.29 : BOOL;
	bArm2VertStn6SpSlanted_30 AT %MX26124.30 : BOOL;
	bArm2VertStn6SpSlanted_31 AT %MX26124.31 : BOOL;

	bArm2VertStn7SpSlanted_00 AT %MX26128.0 : BOOL;
	bArm2VertStn7SpSlanted_01 AT %MX26128.1 : BOOL;
	bArm2VertStn7SpSlanted_02 AT %MX26128.2 : BOOL;
	bArm2VertStn7SpSlanted_03 AT %MX26128.3 : BOOL;
	bArm2VertStn7SpSlanted_04 AT %MX26128.4 : BOOL;
	bArm2VertStn7SpSlanted_05 AT %MX26128.5 : BOOL;
	bArm2VertStn7SpSlanted_06 AT %MX26128.6 : BOOL;
	bArm2VertStn7SpSlanted_07 AT %MX26128.7 : BOOL;
	bArm2VertStn7SpSlanted_08 AT %MX26128.8 : BOOL;
	bArm2VertStn7SpSlanted_09 AT %MX26128.9 : BOOL;
	bArm2VertStn7SpSlanted_10 AT %MX26128.10 : BOOL;
	bArm2VertStn7SpSlanted_11 AT %MX26128.11 : BOOL;
	bArm2VertStn7SpSlanted_12 AT %MX26128.12 : BOOL;
	bArm2VertStn7SpSlanted_13 AT %MX26128.13 : BOOL;
	bArm2VertStn7SpSlanted_14 AT %MX26128.14 : BOOL;
	bArm2VertStn7SpSlanted_15 AT %MX26128.15 : BOOL;
	bArm2VertStn7SpSlanted_16 AT %MX26128.16 : BOOL;
	bArm2VertStn7SpSlanted_17 AT %MX26128.17 : BOOL;
	bArm2VertStn7SpSlanted_18 AT %MX26128.18 : BOOL;
	bArm2VertStn7SpSlanted_19 AT %MX26128.19 : BOOL;
	bArm2VertStn7SpSlanted_20 AT %MX26128.20 : BOOL;
	bArm2VertStn7SpSlanted_21 AT %MX26128.21 : BOOL;
	bArm2VertStn7SpSlanted_22 AT %MX26128.22 : BOOL;
	bArm2VertStn7SpSlanted_23 AT %MX26128.23 : BOOL;
	bArm2VertStn7SpSlanted_24 AT %MX26128.24 : BOOL;
	bArm2VertStn7SpSlanted_25 AT %MX26128.25 : BOOL;
	bArm2VertStn7SpSlanted_26 AT %MX26128.26 : BOOL;
	bArm2VertStn7SpSlanted_27 AT %MX26128.27 : BOOL;
	bArm2VertStn7SpSlanted_28 AT %MX26128.28 : BOOL;
	bArm2VertStn7SpSlanted_29 AT %MX26128.29 : BOOL;
	bArm2VertStn7SpSlanted_30 AT %MX26128.30 : BOOL;
	bArm2VertStn7SpSlanted_31 AT %MX26128.31 : BOOL;

	bArm2VertStn8SpSlanted_00 AT %MX26132.0 : BOOL;
	bArm2VertStn8SpSlanted_01 AT %MX26132.1 : BOOL;
	bArm2VertStn8SpSlanted_02 AT %MX26132.2 : BOOL;
	bArm2VertStn8SpSlanted_03 AT %MX26132.3 : BOOL;
	bArm2VertStn8SpSlanted_04 AT %MX26132.4 : BOOL;
	bArm2VertStn8SpSlanted_05 AT %MX26132.5 : BOOL;
	bArm2VertStn8SpSlanted_06 AT %MX26132.6 : BOOL;
	bArm2VertStn8SpSlanted_07 AT %MX26132.7 : BOOL;
	bArm2VertStn8SpSlanted_08 AT %MX26132.8 : BOOL;
	bArm2VertStn8SpSlanted_09 AT %MX26132.9 : BOOL;
	bArm2VertStn8SpSlanted_10 AT %MX26132.10 : BOOL;
	bArm2VertStn8SpSlanted_11 AT %MX26132.11 : BOOL;
	bArm2VertStn8SpSlanted_12 AT %MX26132.12 : BOOL;
	bArm2VertStn8SpSlanted_13 AT %MX26132.13 : BOOL;
	bArm2VertStn8SpSlanted_14 AT %MX26132.14 : BOOL;
	bArm2VertStn8SpSlanted_15 AT %MX26132.15 : BOOL;
	bArm2VertStn8SpSlanted_16 AT %MX26132.16 : BOOL;
	bArm2VertStn8SpSlanted_17 AT %MX26132.17 : BOOL;
	bArm2VertStn8SpSlanted_18 AT %MX26132.18 : BOOL;
	bArm2VertStn8SpSlanted_19 AT %MX26132.19 : BOOL;
	bArm2VertStn8SpSlanted_20 AT %MX26132.20 : BOOL;
	bArm2VertStn8SpSlanted_21 AT %MX26132.21 : BOOL;
	bArm2VertStn8SpSlanted_22 AT %MX26132.22 : BOOL;
	bArm2VertStn8SpSlanted_23 AT %MX26132.23 : BOOL;
	bArm2VertStn8SpSlanted_24 AT %MX26132.24 : BOOL;
	bArm2VertStn8SpSlanted_25 AT %MX26132.25 : BOOL;
	bArm2VertStn8SpSlanted_26 AT %MX26132.26 : BOOL;
	bArm2VertStn8SpSlanted_27 AT %MX26132.27 : BOOL;
	bArm2VertStn8SpSlanted_28 AT %MX26132.28 : BOOL;
	bArm2VertStn8SpSlanted_29 AT %MX26132.29 : BOOL;
	bArm2VertStn8SpSlanted_30 AT %MX26132.30 : BOOL;
	bArm2VertStn8SpSlanted_31 AT %MX26132.31 : BOOL;

	bArm2VertStn9SpSlanted_00 AT %MX26136.0 : BOOL;
	bArm2VertStn9SpSlanted_01 AT %MX26136.1 : BOOL;
	bArm2VertStn9SpSlanted_02 AT %MX26136.2 : BOOL;
	bArm2VertStn9SpSlanted_03 AT %MX26136.3 : BOOL;
	bArm2VertStn9SpSlanted_04 AT %MX26136.4 : BOOL;
	bArm2VertStn9SpSlanted_05 AT %MX26136.5 : BOOL;
	bArm2VertStn9SpSlanted_06 AT %MX26136.6 : BOOL;
	bArm2VertStn9SpSlanted_07 AT %MX26136.7 : BOOL;
	bArm2VertStn9SpSlanted_08 AT %MX26136.8 : BOOL;
	bArm2VertStn9SpSlanted_09 AT %MX26136.9 : BOOL;
	bArm2VertStn9SpSlanted_10 AT %MX26136.10 : BOOL;
	bArm2VertStn9SpSlanted_11 AT %MX26136.11 : BOOL;
	bArm2VertStn9SpSlanted_12 AT %MX26136.12 : BOOL;
	bArm2VertStn9SpSlanted_13 AT %MX26136.13 : BOOL;
	bArm2VertStn9SpSlanted_14 AT %MX26136.14 : BOOL;
	bArm2VertStn9SpSlanted_15 AT %MX26136.15 : BOOL;
	bArm2VertStn9SpSlanted_16 AT %MX26136.16 : BOOL;
	bArm2VertStn9SpSlanted_17 AT %MX26136.17 : BOOL;
	bArm2VertStn9SpSlanted_18 AT %MX26136.18 : BOOL;
	bArm2VertStn9SpSlanted_19 AT %MX26136.19 : BOOL;
	bArm2VertStn9SpSlanted_20 AT %MX26136.20 : BOOL;
	bArm2VertStn9SpSlanted_21 AT %MX26136.21 : BOOL;
	bArm2VertStn9SpSlanted_22 AT %MX26136.22 : BOOL;
	bArm2VertStn9SpSlanted_23 AT %MX26136.23 : BOOL;
	bArm2VertStn9SpSlanted_24 AT %MX26136.24 : BOOL;
	bArm2VertStn9SpSlanted_25 AT %MX26136.25 : BOOL;
	bArm2VertStn9SpSlanted_26 AT %MX26136.26 : BOOL;
	bArm2VertStn9SpSlanted_27 AT %MX26136.27 : BOOL;
	bArm2VertStn9SpSlanted_28 AT %MX26136.28 : BOOL;
	bArm2VertStn9SpSlanted_29 AT %MX26136.29 : BOOL;
	bArm2VertStn9SpSlanted_30 AT %MX26136.30 : BOOL;
	bArm2VertStn9SpSlanted_31 AT %MX26136.31 : BOOL;

	bArm2VertStn10SpSlanted_00 AT %MX26140.0 : BOOL;
	bArm2VertStn10SpSlanted_01 AT %MX26140.1 : BOOL;
	bArm2VertStn10SpSlanted_02 AT %MX26140.2 : BOOL;
	bArm2VertStn10SpSlanted_03 AT %MX26140.3 : BOOL;
	bArm2VertStn10SpSlanted_04 AT %MX26140.4 : BOOL;
	bArm2VertStn10SpSlanted_05 AT %MX26140.5 : BOOL;
	bArm2VertStn10SpSlanted_06 AT %MX26140.6 : BOOL;
	bArm2VertStn10SpSlanted_07 AT %MX26140.7 : BOOL;
	bArm2VertStn10SpSlanted_08 AT %MX26140.8 : BOOL;
	bArm2VertStn10SpSlanted_09 AT %MX26140.9 : BOOL;
	bArm2VertStn10SpSlanted_10 AT %MX26140.10 : BOOL;
	bArm2VertStn10SpSlanted_11 AT %MX26140.11 : BOOL;
	bArm2VertStn10SpSlanted_12 AT %MX26140.12 : BOOL;
	bArm2VertStn10SpSlanted_13 AT %MX26140.13 : BOOL;
	bArm2VertStn10SpSlanted_14 AT %MX26140.14 : BOOL;
	bArm2VertStn10SpSlanted_15 AT %MX26140.15 : BOOL;
	bArm2VertStn10SpSlanted_16 AT %MX26140.16 : BOOL;
	bArm2VertStn10SpSlanted_17 AT %MX26140.17 : BOOL;
	bArm2VertStn10SpSlanted_18 AT %MX26140.18 : BOOL;
	bArm2VertStn10SpSlanted_19 AT %MX26140.19 : BOOL;
	bArm2VertStn10SpSlanted_20 AT %MX26140.20 : BOOL;
	bArm2VertStn10SpSlanted_21 AT %MX26140.21 : BOOL;
	bArm2VertStn10SpSlanted_22 AT %MX26140.22 : BOOL;
	bArm2VertStn10SpSlanted_23 AT %MX26140.23 : BOOL;
	bArm2VertStn10SpSlanted_24 AT %MX26140.24 : BOOL;
	bArm2VertStn10SpSlanted_25 AT %MX26140.25 : BOOL;
	bArm2VertStn10SpSlanted_26 AT %MX26140.26 : BOOL;
	bArm2VertStn10SpSlanted_27 AT %MX26140.27 : BOOL;
	bArm2VertStn10SpSlanted_28 AT %MX26140.28 : BOOL;
	bArm2VertStn10SpSlanted_29 AT %MX26140.29 : BOOL;
	bArm2VertStn10SpSlanted_30 AT %MX26140.30 : BOOL;
	bArm2VertStn10SpSlanted_31 AT %MX26140.31 : BOOL;

	bArm2VertStn11SpSlanted_00 AT %MX26144.0 : BOOL;
	bArm2VertStn11SpSlanted_01 AT %MX26144.1 : BOOL;
	bArm2VertStn11SpSlanted_02 AT %MX26144.2 : BOOL;
	bArm2VertStn11SpSlanted_03 AT %MX26144.3 : BOOL;
	bArm2VertStn11SpSlanted_04 AT %MX26144.4 : BOOL;
	bArm2VertStn11SpSlanted_05 AT %MX26144.5 : BOOL;
	bArm2VertStn11SpSlanted_06 AT %MX26144.6 : BOOL;
	bArm2VertStn11SpSlanted_07 AT %MX26144.7 : BOOL;
	bArm2VertStn11SpSlanted_08 AT %MX26144.8 : BOOL;
	bArm2VertStn11SpSlanted_09 AT %MX26144.9 : BOOL;
	bArm2VertStn11SpSlanted_10 AT %MX26144.10 : BOOL;
	bArm2VertStn11SpSlanted_11 AT %MX26144.11 : BOOL;
	bArm2VertStn11SpSlanted_12 AT %MX26144.12 : BOOL;
	bArm2VertStn11SpSlanted_13 AT %MX26144.13 : BOOL;
	bArm2VertStn11SpSlanted_14 AT %MX26144.14 : BOOL;
	bArm2VertStn11SpSlanted_15 AT %MX26144.15 : BOOL;
	bArm2VertStn11SpSlanted_16 AT %MX26144.16 : BOOL;
	bArm2VertStn11SpSlanted_17 AT %MX26144.17 : BOOL;
	bArm2VertStn11SpSlanted_18 AT %MX26144.18 : BOOL;
	bArm2VertStn11SpSlanted_19 AT %MX26144.19 : BOOL;
	bArm2VertStn11SpSlanted_20 AT %MX26144.20 : BOOL;
	bArm2VertStn11SpSlanted_21 AT %MX26144.21 : BOOL;
	bArm2VertStn11SpSlanted_22 AT %MX26144.22 : BOOL;
	bArm2VertStn11SpSlanted_23 AT %MX26144.23 : BOOL;
	bArm2VertStn11SpSlanted_24 AT %MX26144.24 : BOOL;
	bArm2VertStn11SpSlanted_25 AT %MX26144.25 : BOOL;
	bArm2VertStn11SpSlanted_26 AT %MX26144.26 : BOOL;
	bArm2VertStn11SpSlanted_27 AT %MX26144.27 : BOOL;
	bArm2VertStn11SpSlanted_28 AT %MX26144.28 : BOOL;
	bArm2VertStn11SpSlanted_29 AT %MX26144.29 : BOOL;
	bArm2VertStn11SpSlanted_30 AT %MX26144.30 : BOOL;
	bArm2VertStn11SpSlanted_31 AT %MX26144.31 : BOOL;

	bArm2VertStn12SpSlanted_00 AT %MX26148.0 : BOOL;
	bArm2VertStn12SpSlanted_01 AT %MX26148.1 : BOOL;
	bArm2VertStn12SpSlanted_02 AT %MX26148.2 : BOOL;
	bArm2VertStn12SpSlanted_03 AT %MX26148.3 : BOOL;
	bArm2VertStn12SpSlanted_04 AT %MX26148.4 : BOOL;
	bArm2VertStn12SpSlanted_05 AT %MX26148.5 : BOOL;
	bArm2VertStn12SpSlanted_06 AT %MX26148.6 : BOOL;
	bArm2VertStn12SpSlanted_07 AT %MX26148.7 : BOOL;
	bArm2VertStn12SpSlanted_08 AT %MX26148.8 : BOOL;
	bArm2VertStn12SpSlanted_09 AT %MX26148.9 : BOOL;
	bArm2VertStn12SpSlanted_10 AT %MX26148.10 : BOOL;
	bArm2VertStn12SpSlanted_11 AT %MX26148.11 : BOOL;
	bArm2VertStn12SpSlanted_12 AT %MX26148.12 : BOOL;
	bArm2VertStn12SpSlanted_13 AT %MX26148.13 : BOOL;
	bArm2VertStn12SpSlanted_14 AT %MX26148.14 : BOOL;
	bArm2VertStn12SpSlanted_15 AT %MX26148.15 : BOOL;
	bArm2VertStn12SpSlanted_16 AT %MX26148.16 : BOOL;
	bArm2VertStn12SpSlanted_17 AT %MX26148.17 : BOOL;
	bArm2VertStn12SpSlanted_18 AT %MX26148.18 : BOOL;
	bArm2VertStn12SpSlanted_19 AT %MX26148.19 : BOOL;
	bArm2VertStn12SpSlanted_20 AT %MX26148.20 : BOOL;
	bArm2VertStn12SpSlanted_21 AT %MX26148.21 : BOOL;
	bArm2VertStn12SpSlanted_22 AT %MX26148.22 : BOOL;
	bArm2VertStn12SpSlanted_23 AT %MX26148.23 : BOOL;
	bArm2VertStn12SpSlanted_24 AT %MX26148.24 : BOOL;
	bArm2VertStn12SpSlanted_25 AT %MX26148.25 : BOOL;
	bArm2VertStn12SpSlanted_26 AT %MX26148.26 : BOOL;
	bArm2VertStn12SpSlanted_27 AT %MX26148.27 : BOOL;
	bArm2VertStn12SpSlanted_28 AT %MX26148.28 : BOOL;
	bArm2VertStn12SpSlanted_29 AT %MX26148.29 : BOOL;
	bArm2VertStn12SpSlanted_30 AT %MX26148.30 : BOOL;
	bArm2VertStn12SpSlanted_31 AT %MX26148.31 : BOOL;


(* xxxxxxxxxxxxxxxxxxxxxxxxxxxxxxxxxxxxxxx Vert xxxxxxxxxxxxxxxxxxxxxxxxxxxxxxxxxxxxxxx*)
(*========= Down Regular BOOL LINK with %MX26200-MX26299 =========*)

	bArm2VertStn1Regular_00 AT %MX26204.0 : BOOL;
	bArm2VertStn1Regular_01 AT %MX26204.1 : BOOL;
	bArm2VertStn1Regular_02 AT %MX26204.2 : BOOL;
	bArm2VertStn1Regular_03 AT %MX26204.3 : BOOL;
	bArm2VertStn1Regular_04 AT %MX26204.4 : BOOL;
	bArm2VertStn1Regular_05 AT %MX26204.5 : BOOL;
	bArm2VertStn1Regular_06 AT %MX26204.6 : BOOL;
	bArm2VertStn1Regular_07 AT %MX26204.7 : BOOL;
	bArm2VertStn1Regular_08 AT %MX26204.8 : BOOL;
	bArm2VertStn1Regular_09 AT %MX26204.9 : BOOL;
	bArm2VertStn1Regular_10 AT %MX26204.10 : BOOL;
	bArm2VertStn1Regular_11 AT %MX26204.11 : BOOL;
	bArm2VertStn1Regular_12 AT %MX26204.12 : BOOL;
	bArm2VertStn1Regular_13 AT %MX26204.13 : BOOL;
	bArm2VertStn1Regular_14 AT %MX26204.14 : BOOL;
	bArm2VertStn1Regular_15 AT %MX26204.15 : BOOL;
	bArm2VertStn1Regular_16 AT %MX26204.16 : BOOL;
	bArm2VertStn1Regular_17 AT %MX26204.17 : BOOL;
	bArm2VertStn1Regular_18 AT %MX26204.18 : BOOL;
	bArm2VertStn1Regular_19 AT %MX26204.19 : BOOL;
	bArm2VertStn1Regular_20 AT %MX26204.20 : BOOL;
	bArm2VertStn1Regular_21 AT %MX26204.21 : BOOL;
	bArm2VertStn1Regular_22 AT %MX26204.22 : BOOL;
	bArm2VertStn1Regular_23 AT %MX26204.23 : BOOL;
	bArm2VertStn1Regular_24 AT %MX26204.24 : BOOL;
	bArm2VertStn1Regular_25 AT %MX26204.25 : BOOL;
	bArm2VertStn1Regular_26 AT %MX26204.26 : BOOL;
	bArm2VertStn1Regular_27 AT %MX26204.27 : BOOL;
	bArm2VertStn1Regular_28 AT %MX26204.28 : BOOL;
	bArm2VertStn1Regular_29 AT %MX26204.29 : BOOL;
	bArm2VertStn1Regular_30 AT %MX26204.30 : BOOL;
	bArm2VertStn1Regular_31 AT %MX26204.31 : BOOL;

	bArm2VertStn2Regular_00 AT %MX26208.0 : BOOL;
	bArm2VertStn2Regular_01 AT %MX26208.1 : BOOL;
	bArm2VertStn2Regular_02 AT %MX26208.2 : BOOL;
	bArm2VertStn2Regular_03 AT %MX26208.3 : BOOL;
	bArm2VertStn2Regular_04 AT %MX26208.4 : BOOL;
	bArm2VertStn2Regular_05 AT %MX26208.5 : BOOL;
	bArm2VertStn2Regular_06 AT %MX26208.6 : BOOL;
	bArm2VertStn2Regular_07 AT %MX26208.7 : BOOL;
	bArm2VertStn2Regular_08 AT %MX26208.8 : BOOL;
	bArm2VertStn2Regular_09 AT %MX26208.9 : BOOL;
	bArm2VertStn2Regular_10 AT %MX26208.10 : BOOL;
	bArm2VertStn2Regular_11 AT %MX26208.11 : BOOL;
	bArm2VertStn2Regular_12 AT %MX26208.12 : BOOL;
	bArm2VertStn2Regular_13 AT %MX26208.13 : BOOL;
	bArm2VertStn2Regular_14 AT %MX26208.14 : BOOL;
	bArm2VertStn2Regular_15 AT %MX26208.15 : BOOL;
	bArm2VertStn2Regular_16 AT %MX26208.16 : BOOL;
	bArm2VertStn2Regular_17 AT %MX26208.17 : BOOL;
	bArm2VertStn2Regular_18 AT %MX26208.18 : BOOL;
	bArm2VertStn2Regular_19 AT %MX26208.19 : BOOL;
	bArm2VertStn2Regular_20 AT %MX26208.20 : BOOL;
	bArm2VertStn2Regular_21 AT %MX26208.21 : BOOL;
	bArm2VertStn2Regular_22 AT %MX26208.22 : BOOL;
	bArm2VertStn2Regular_23 AT %MX26208.23 : BOOL;
	bArm2VertStn2Regular_24 AT %MX26208.24 : BOOL;
	bArm2VertStn2Regular_25 AT %MX26208.25 : BOOL;
	bArm2VertStn2Regular_26 AT %MX26208.26 : BOOL;
	bArm2VertStn2Regular_27 AT %MX26208.27 : BOOL;
	bArm2VertStn2Regular_28 AT %MX26208.28 : BOOL;
	bArm2VertStn2Regular_29 AT %MX26208.29 : BOOL;
	bArm2VertStn2Regular_30 AT %MX26208.30 : BOOL;
	bArm2VertStn2Regular_31 AT %MX26208.31 : BOOL;

	bArm2VertStn3Regular_00 AT %MX26212.0 : BOOL;
	bArm2VertStn3Regular_01 AT %MX26212.1 : BOOL;
	bArm2VertStn3Regular_02 AT %MX26212.2 : BOOL;
	bArm2VertStn3Regular_03 AT %MX26212.3 : BOOL;
	bArm2VertStn3Regular_04 AT %MX26212.4 : BOOL;
	bArm2VertStn3Regular_05 AT %MX26212.5 : BOOL;
	bArm2VertStn3Regular_06 AT %MX26212.6 : BOOL;
	bArm2VertStn3Regular_07 AT %MX26212.7 : BOOL;
	bArm2VertStn3Regular_08 AT %MX26212.8 : BOOL;
	bArm2VertStn3Regular_09 AT %MX26212.9 : BOOL;
	bArm2VertStn3Regular_10 AT %MX26212.10 : BOOL;
	bArm2VertStn3Regular_11 AT %MX26212.11 : BOOL;
	bArm2VertStn3Regular_12 AT %MX26212.12 : BOOL;
	bArm2VertStn3Regular_13 AT %MX26212.13 : BOOL;
	bArm2VertStn3Regular_14 AT %MX26212.14 : BOOL;
	bArm2VertStn3Regular_15 AT %MX26212.15 : BOOL;
	bArm2VertStn3Regular_16 AT %MX26212.16 : BOOL;
	bArm2VertStn3Regular_17 AT %MX26212.17 : BOOL;
	bArm2VertStn3Regular_18 AT %MX26212.18 : BOOL;
	bArm2VertStn3Regular_19 AT %MX26212.19 : BOOL;
	bArm2VertStn3Regular_20 AT %MX26212.20 : BOOL;
	bArm2VertStn3Regular_21 AT %MX26212.21 : BOOL;
	bArm2VertStn3Regular_22 AT %MX26212.22 : BOOL;
	bArm2VertStn3Regular_23 AT %MX26212.23 : BOOL;
	bArm2VertStn3Regular_24 AT %MX26212.24 : BOOL;
	bArm2VertStn3Regular_25 AT %MX26212.25 : BOOL;
	bArm2VertStn3Regular_26 AT %MX26212.26 : BOOL;
	bArm2VertStn3Regular_27 AT %MX26212.27 : BOOL;
	bArm2VertStn3Regular_28 AT %MX26212.28 : BOOL;
	bArm2VertStn3Regular_29 AT %MX26212.29 : BOOL;
	bArm2VertStn3Regular_30 AT %MX26212.30 : BOOL;
	bArm2VertStn3Regular_31 AT %MX26212.31 : BOOL;

	bArm2VertStn4Regular_00 AT %MX26216.0 : BOOL;
	bArm2VertStn4Regular_01 AT %MX26216.1 : BOOL;
	bArm2VertStn4Regular_02 AT %MX26216.2 : BOOL;
	bArm2VertStn4Regular_03 AT %MX26216.3 : BOOL;
	bArm2VertStn4Regular_04 AT %MX26216.4 : BOOL;
	bArm2VertStn4Regular_05 AT %MX26216.5 : BOOL;
	bArm2VertStn4Regular_06 AT %MX26216.6 : BOOL;
	bArm2VertStn4Regular_07 AT %MX26216.7 : BOOL;
	bArm2VertStn4Regular_08 AT %MX26216.8 : BOOL;
	bArm2VertStn4Regular_09 AT %MX26216.9 : BOOL;
	bArm2VertStn4Regular_10 AT %MX26216.10 : BOOL;
	bArm2VertStn4Regular_11 AT %MX26216.11 : BOOL;
	bArm2VertStn4Regular_12 AT %MX26216.12 : BOOL;
	bArm2VertStn4Regular_13 AT %MX26216.13 : BOOL;
	bArm2VertStn4Regular_14 AT %MX26216.14 : BOOL;
	bArm2VertStn4Regular_15 AT %MX26216.15 : BOOL;
	bArm2VertStn4Regular_16 AT %MX26216.16 : BOOL;
	bArm2VertStn4Regular_17 AT %MX26216.17 : BOOL;
	bArm2VertStn4Regular_18 AT %MX26216.18 : BOOL;
	bArm2VertStn4Regular_19 AT %MX26216.19 : BOOL;
	bArm2VertStn4Regular_20 AT %MX26216.20 : BOOL;
	bArm2VertStn4Regular_21 AT %MX26216.21 : BOOL;
	bArm2VertStn4Regular_22 AT %MX26216.22 : BOOL;
	bArm2VertStn4Regular_23 AT %MX26216.23 : BOOL;
	bArm2VertStn4Regular_24 AT %MX26216.24 : BOOL;
	bArm2VertStn4Regular_25 AT %MX26216.25 : BOOL;
	bArm2VertStn4Regular_26 AT %MX26216.26 : BOOL;
	bArm2VertStn4Regular_27 AT %MX26216.27 : BOOL;
	bArm2VertStn4Regular_28 AT %MX26216.28 : BOOL;
	bArm2VertStn4Regular_29 AT %MX26216.29 : BOOL;
	bArm2VertStn4Regular_30 AT %MX26216.30 : BOOL;
	bArm2VertStn4Regular_31 AT %MX26216.31 : BOOL;

	bArm2VertStn5Regular_00 AT %MX26220.0 : BOOL;
	bArm2VertStn5Regular_01 AT %MX26220.1 : BOOL;
	bArm2VertStn5Regular_02 AT %MX26220.2 : BOOL;
	bArm2VertStn5Regular_03 AT %MX26220.3 : BOOL;
	bArm2VertStn5Regular_04 AT %MX26220.4 : BOOL;
	bArm2VertStn5Regular_05 AT %MX26220.5 : BOOL;
	bArm2VertStn5Regular_06 AT %MX26220.6 : BOOL;
	bArm2VertStn5Regular_07 AT %MX26220.7 : BOOL;
	bArm2VertStn5Regular_08 AT %MX26220.8 : BOOL;
	bArm2VertStn5Regular_09 AT %MX26220.9 : BOOL;
	bArm2VertStn5Regular_10 AT %MX26220.10 : BOOL;
	bArm2VertStn5Regular_11 AT %MX26220.11 : BOOL;
	bArm2VertStn5Regular_12 AT %MX26220.12 : BOOL;
	bArm2VertStn5Regular_13 AT %MX26220.13 : BOOL;
	bArm2VertStn5Regular_14 AT %MX26220.14 : BOOL;
	bArm2VertStn5Regular_15 AT %MX26220.15 : BOOL;
	bArm2VertStn5Regular_16 AT %MX26220.16 : BOOL;
	bArm2VertStn5Regular_17 AT %MX26220.17 : BOOL;
	bArm2VertStn5Regular_18 AT %MX26220.18 : BOOL;
	bArm2VertStn5Regular_19 AT %MX26220.19 : BOOL;
	bArm2VertStn5Regular_20 AT %MX26220.20 : BOOL;
	bArm2VertStn5Regular_21 AT %MX26220.21 : BOOL;
	bArm2VertStn5Regular_22 AT %MX26220.22 : BOOL;
	bArm2VertStn5Regular_23 AT %MX26220.23 : BOOL;
	bArm2VertStn5Regular_24 AT %MX26220.24 : BOOL;
	bArm2VertStn5Regular_25 AT %MX26220.25 : BOOL;
	bArm2VertStn5Regular_26 AT %MX26220.26 : BOOL;
	bArm2VertStn5Regular_27 AT %MX26220.27 : BOOL;
	bArm2VertStn5Regular_28 AT %MX26220.28 : BOOL;
	bArm2VertStn5Regular_29 AT %MX26220.29 : BOOL;
	bArm2VertStn5Regular_30 AT %MX26220.30 : BOOL;
	bArm2VertStn5Regular_31 AT %MX26220.31 : BOOL;

	bArm2VertStn6Regular_00 AT %MX26224.0 : BOOL;
	bArm2VertStn6Regular_01 AT %MX26224.1 : BOOL;
	bArm2VertStn6Regular_02 AT %MX26224.2 : BOOL;
	bArm2VertStn6Regular_03 AT %MX26224.3 : BOOL;
	bArm2VertStn6Regular_04 AT %MX26224.4 : BOOL;
	bArm2VertStn6Regular_05 AT %MX26224.5 : BOOL;
	bArm2VertStn6Regular_06 AT %MX26224.6 : BOOL;
	bArm2VertStn6Regular_07 AT %MX26224.7 : BOOL;
	bArm2VertStn6Regular_08 AT %MX26224.8 : BOOL;
	bArm2VertStn6Regular_09 AT %MX26224.9 : BOOL;
	bArm2VertStn6Regular_10 AT %MX26224.10 : BOOL;
	bArm2VertStn6Regular_11 AT %MX26224.11 : BOOL;
	bArm2VertStn6Regular_12 AT %MX26224.12 : BOOL;
	bArm2VertStn6Regular_13 AT %MX26224.13 : BOOL;
	bArm2VertStn6Regular_14 AT %MX26224.14 : BOOL;
	bArm2VertStn6Regular_15 AT %MX26224.15 : BOOL;
	bArm2VertStn6Regular_16 AT %MX26224.16 : BOOL;
	bArm2VertStn6Regular_17 AT %MX26224.17 : BOOL;
	bArm2VertStn6Regular_18 AT %MX26224.18 : BOOL;
	bArm2VertStn6Regular_19 AT %MX26224.19 : BOOL;
	bArm2VertStn6Regular_20 AT %MX26224.20 : BOOL;
	bArm2VertStn6Regular_21 AT %MX26224.21 : BOOL;
	bArm2VertStn6Regular_22 AT %MX26224.22 : BOOL;
	bArm2VertStn6Regular_23 AT %MX26224.23 : BOOL;
	bArm2VertStn6Regular_24 AT %MX26224.24 : BOOL;
	bArm2VertStn6Regular_25 AT %MX26224.25 : BOOL;
	bArm2VertStn6Regular_26 AT %MX26224.26 : BOOL;
	bArm2VertStn6Regular_27 AT %MX26224.27 : BOOL;
	bArm2VertStn6Regular_28 AT %MX26224.28 : BOOL;
	bArm2VertStn6Regular_29 AT %MX26224.29 : BOOL;
	bArm2VertStn6Regular_30 AT %MX26224.30 : BOOL;
	bArm2VertStn6Regular_31 AT %MX26224.31 : BOOL;

	bArm2VertStn7Regular_00 AT %MX26228.0 : BOOL;
	bArm2VertStn7Regular_01 AT %MX26228.1 : BOOL;
	bArm2VertStn7Regular_02 AT %MX26228.2 : BOOL;
	bArm2VertStn7Regular_03 AT %MX26228.3 : BOOL;
	bArm2VertStn7Regular_04 AT %MX26228.4 : BOOL;
	bArm2VertStn7Regular_05 AT %MX26228.5 : BOOL;
	bArm2VertStn7Regular_06 AT %MX26228.6 : BOOL;
	bArm2VertStn7Regular_07 AT %MX26228.7 : BOOL;
	bArm2VertStn7Regular_08 AT %MX26228.8 : BOOL;
	bArm2VertStn7Regular_09 AT %MX26228.9 : BOOL;
	bArm2VertStn7Regular_10 AT %MX26228.10 : BOOL;
	bArm2VertStn7Regular_11 AT %MX26228.11 : BOOL;
	bArm2VertStn7Regular_12 AT %MX26228.12 : BOOL;
	bArm2VertStn7Regular_13 AT %MX26228.13 : BOOL;
	bArm2VertStn7Regular_14 AT %MX26228.14 : BOOL;
	bArm2VertStn7Regular_15 AT %MX26228.15 : BOOL;
	bArm2VertStn7Regular_16 AT %MX26228.16 : BOOL;
	bArm2VertStn7Regular_17 AT %MX26228.17 : BOOL;
	bArm2VertStn7Regular_18 AT %MX26228.18 : BOOL;
	bArm2VertStn7Regular_19 AT %MX26228.19 : BOOL;
	bArm2VertStn7Regular_20 AT %MX26228.20 : BOOL;
	bArm2VertStn7Regular_21 AT %MX26228.21 : BOOL;
	bArm2VertStn7Regular_22 AT %MX26228.22 : BOOL;
	bArm2VertStn7Regular_23 AT %MX26228.23 : BOOL;
	bArm2VertStn7Regular_24 AT %MX26228.24 : BOOL;
	bArm2VertStn7Regular_25 AT %MX26228.25 : BOOL;
	bArm2VertStn7Regular_26 AT %MX26228.26 : BOOL;
	bArm2VertStn7Regular_27 AT %MX26228.27 : BOOL;
	bArm2VertStn7Regular_28 AT %MX26228.28 : BOOL;
	bArm2VertStn7Regular_29 AT %MX26228.29 : BOOL;
	bArm2VertStn7Regular_30 AT %MX26228.30 : BOOL;
	bArm2VertStn7Regular_31 AT %MX26228.31 : BOOL;

	bArm2VertStn8Regular_00 AT %MX26232.0 : BOOL;
	bArm2VertStn8Regular_01 AT %MX26232.1 : BOOL;
	bArm2VertStn8Regular_02 AT %MX26232.2 : BOOL;
	bArm2VertStn8Regular_03 AT %MX26232.3 : BOOL;
	bArm2VertStn8Regular_04 AT %MX26232.4 : BOOL;
	bArm2VertStn8Regular_05 AT %MX26232.5 : BOOL;
	bArm2VertStn8Regular_06 AT %MX26232.6 : BOOL;
	bArm2VertStn8Regular_07 AT %MX26232.7 : BOOL;
	bArm2VertStn8Regular_08 AT %MX26232.8 : BOOL;
	bArm2VertStn8Regular_09 AT %MX26232.9 : BOOL;
	bArm2VertStn8Regular_10 AT %MX26232.10 : BOOL;
	bArm2VertStn8Regular_11 AT %MX26232.11 : BOOL;
	bArm2VertStn8Regular_12 AT %MX26232.12 : BOOL;
	bArm2VertStn8Regular_13 AT %MX26232.13 : BOOL;
	bArm2VertStn8Regular_14 AT %MX26232.14 : BOOL;
	bArm2VertStn8Regular_15 AT %MX26232.15 : BOOL;
	bArm2VertStn8Regular_16 AT %MX26232.16 : BOOL;
	bArm2VertStn8Regular_17 AT %MX26232.17 : BOOL;
	bArm2VertStn8Regular_18 AT %MX26232.18 : BOOL;
	bArm2VertStn8Regular_19 AT %MX26232.19 : BOOL;
	bArm2VertStn8Regular_20 AT %MX26232.20 : BOOL;
	bArm2VertStn8Regular_21 AT %MX26232.21 : BOOL;
	bArm2VertStn8Regular_22 AT %MX26232.22 : BOOL;
	bArm2VertStn8Regular_23 AT %MX26232.23 : BOOL;
	bArm2VertStn8Regular_24 AT %MX26232.24 : BOOL;
	bArm2VertStn8Regular_25 AT %MX26232.25 : BOOL;
	bArm2VertStn8Regular_26 AT %MX26232.26 : BOOL;
	bArm2VertStn8Regular_27 AT %MX26232.27 : BOOL;
	bArm2VertStn8Regular_28 AT %MX26232.28 : BOOL;
	bArm2VertStn8Regular_29 AT %MX26232.29 : BOOL;
	bArm2VertStn8Regular_30 AT %MX26232.30 : BOOL;
	bArm2VertStn8Regular_31 AT %MX26232.31 : BOOL;

	bArm2VertStn9Regular_00 AT %MX26236.0 : BOOL;
	bArm2VertStn9Regular_01 AT %MX26236.1 : BOOL;
	bArm2VertStn9Regular_02 AT %MX26236.2 : BOOL;
	bArm2VertStn9Regular_03 AT %MX26236.3 : BOOL;
	bArm2VertStn9Regular_04 AT %MX26236.4 : BOOL;
	bArm2VertStn9Regular_05 AT %MX26236.5 : BOOL;
	bArm2VertStn9Regular_06 AT %MX26236.6 : BOOL;
	bArm2VertStn9Regular_07 AT %MX26236.7 : BOOL;
	bArm2VertStn9Regular_08 AT %MX26236.8 : BOOL;
	bArm2VertStn9Regular_09 AT %MX26236.9 : BOOL;
	bArm2VertStn9Regular_10 AT %MX26236.10 : BOOL;
	bArm2VertStn9Regular_11 AT %MX26236.11 : BOOL;
	bArm2VertStn9Regular_12 AT %MX26236.12 : BOOL;
	bArm2VertStn9Regular_13 AT %MX26236.13 : BOOL;
	bArm2VertStn9Regular_14 AT %MX26236.14 : BOOL;
	bArm2VertStn9Regular_15 AT %MX26236.15 : BOOL;
	bArm2VertStn9Regular_16 AT %MX26236.16 : BOOL;
	bArm2VertStn9Regular_17 AT %MX26236.17 : BOOL;
	bArm2VertStn9Regular_18 AT %MX26236.18 : BOOL;
	bArm2VertStn9Regular_19 AT %MX26236.19 : BOOL;
	bArm2VertStn9Regular_20 AT %MX26236.20 : BOOL;
	bArm2VertStn9Regular_21 AT %MX26236.21 : BOOL;
	bArm2VertStn9Regular_22 AT %MX26236.22 : BOOL;
	bArm2VertStn9Regular_23 AT %MX26236.23 : BOOL;
	bArm2VertStn9Regular_24 AT %MX26236.24 : BOOL;
	bArm2VertStn9Regular_25 AT %MX26236.25 : BOOL;
	bArm2VertStn9Regular_26 AT %MX26236.26 : BOOL;
	bArm2VertStn9Regular_27 AT %MX26236.27 : BOOL;
	bArm2VertStn9Regular_28 AT %MX26236.28 : BOOL;
	bArm2VertStn9Regular_29 AT %MX26236.29 : BOOL;
	bArm2VertStn9Regular_30 AT %MX26236.30 : BOOL;
	bArm2VertStn9Regular_31 AT %MX26236.31 : BOOL;

	bArm2VertStn10Regular_00 AT %MX26240.0 : BOOL;
	bArm2VertStn10Regular_01 AT %MX26240.1 : BOOL;
	bArm2VertStn10Regular_02 AT %MX26240.2 : BOOL;
	bArm2VertStn10Regular_03 AT %MX26240.3 : BOOL;
	bArm2VertStn10Regular_04 AT %MX26240.4 : BOOL;
	bArm2VertStn10Regular_05 AT %MX26240.5 : BOOL;
	bArm2VertStn10Regular_06 AT %MX26240.6 : BOOL;
	bArm2VertStn10Regular_07 AT %MX26240.7 : BOOL;
	bArm2VertStn10Regular_08 AT %MX26240.8 : BOOL;
	bArm2VertStn10Regular_09 AT %MX26240.9 : BOOL;
	bArm2VertStn10Regular_10 AT %MX26240.10 : BOOL;
	bArm2VertStn10Regular_11 AT %MX26240.11 : BOOL;
	bArm2VertStn10Regular_12 AT %MX26240.12 : BOOL;
	bArm2VertStn10Regular_13 AT %MX26240.13 : BOOL;
	bArm2VertStn10Regular_14 AT %MX26240.14 : BOOL;
	bArm2VertStn10Regular_15 AT %MX26240.15 : BOOL;
	bArm2VertStn10Regular_16 AT %MX26240.16 : BOOL;
	bArm2VertStn10Regular_17 AT %MX26240.17 : BOOL;
	bArm2VertStn10Regular_18 AT %MX26240.18 : BOOL;
	bArm2VertStn10Regular_19 AT %MX26240.19 : BOOL;
	bArm2VertStn10Regular_20 AT %MX26240.20 : BOOL;
	bArm2VertStn10Regular_21 AT %MX26240.21 : BOOL;
	bArm2VertStn10Regular_22 AT %MX26240.22 : BOOL;
	bArm2VertStn10Regular_23 AT %MX26240.23 : BOOL;
	bArm2VertStn10Regular_24 AT %MX26240.24 : BOOL;
	bArm2VertStn10Regular_25 AT %MX26240.25 : BOOL;
	bArm2VertStn10Regular_26 AT %MX26240.26 : BOOL;
	bArm2VertStn10Regular_27 AT %MX26240.27 : BOOL;
	bArm2VertStn10Regular_28 AT %MX26240.28 : BOOL;
	bArm2VertStn10Regular_29 AT %MX26240.29 : BOOL;
	bArm2VertStn10Regular_30 AT %MX26240.30 : BOOL;
	bArm2VertStn10Regular_31 AT %MX26240.31 : BOOL;

	bArm2VertStn11Regular_00 AT %MX26244.0 : BOOL;
	bArm2VertStn11Regular_01 AT %MX26244.1 : BOOL;
	bArm2VertStn11Regular_02 AT %MX26244.2 : BOOL;
	bArm2VertStn11Regular_03 AT %MX26244.3 : BOOL;
	bArm2VertStn11Regular_04 AT %MX26244.4 : BOOL;
	bArm2VertStn11Regular_05 AT %MX26244.5 : BOOL;
	bArm2VertStn11Regular_06 AT %MX26244.6 : BOOL;
	bArm2VertStn11Regular_07 AT %MX26244.7 : BOOL;
	bArm2VertStn11Regular_08 AT %MX26244.8 : BOOL;
	bArm2VertStn11Regular_09 AT %MX26244.9 : BOOL;
	bArm2VertStn11Regular_10 AT %MX26244.10 : BOOL;
	bArm2VertStn11Regular_11 AT %MX26244.11 : BOOL;
	bArm2VertStn11Regular_12 AT %MX26244.12 : BOOL;
	bArm2VertStn11Regular_13 AT %MX26244.13 : BOOL;
	bArm2VertStn11Regular_14 AT %MX26244.14 : BOOL;
	bArm2VertStn11Regular_15 AT %MX26244.15 : BOOL;
	bArm2VertStn11Regular_16 AT %MX26244.16 : BOOL;
	bArm2VertStn11Regular_17 AT %MX26244.17 : BOOL;
	bArm2VertStn11Regular_18 AT %MX26244.18 : BOOL;
	bArm2VertStn11Regular_19 AT %MX26244.19 : BOOL;
	bArm2VertStn11Regular_20 AT %MX26244.20 : BOOL;
	bArm2VertStn11Regular_21 AT %MX26244.21 : BOOL;
	bArm2VertStn11Regular_22 AT %MX26244.22 : BOOL;
	bArm2VertStn11Regular_23 AT %MX26244.23 : BOOL;
	bArm2VertStn11Regular_24 AT %MX26244.24 : BOOL;
	bArm2VertStn11Regular_25 AT %MX26244.25 : BOOL;
	bArm2VertStn11Regular_26 AT %MX26244.26 : BOOL;
	bArm2VertStn11Regular_27 AT %MX26244.27 : BOOL;
	bArm2VertStn11Regular_28 AT %MX26244.28 : BOOL;
	bArm2VertStn11Regular_29 AT %MX26244.29 : BOOL;
	bArm2VertStn11Regular_30 AT %MX26244.30 : BOOL;
	bArm2VertStn11Regular_31 AT %MX26244.31 : BOOL;

	bArm2VertStn12Regular_00 AT %MX26248.0 : BOOL;
	bArm2VertStn12Regular_01 AT %MX26248.1 : BOOL;
	bArm2VertStn12Regular_02 AT %MX26248.2 : BOOL;
	bArm2VertStn12Regular_03 AT %MX26248.3 : BOOL;
	bArm2VertStn12Regular_04 AT %MX26248.4 : BOOL;
	bArm2VertStn12Regular_05 AT %MX26248.5 : BOOL;
	bArm2VertStn12Regular_06 AT %MX26248.6 : BOOL;
	bArm2VertStn12Regular_07 AT %MX26248.7 : BOOL;
	bArm2VertStn12Regular_08 AT %MX26248.8 : BOOL;
	bArm2VertStn12Regular_09 AT %MX26248.9 : BOOL;
	bArm2VertStn12Regular_10 AT %MX26248.10 : BOOL;
	bArm2VertStn12Regular_11 AT %MX26248.11 : BOOL;
	bArm2VertStn12Regular_12 AT %MX26248.12 : BOOL;
	bArm2VertStn12Regular_13 AT %MX26248.13 : BOOL;
	bArm2VertStn12Regular_14 AT %MX26248.14 : BOOL;
	bArm2VertStn12Regular_15 AT %MX26248.15 : BOOL;
	bArm2VertStn12Regular_16 AT %MX26248.16 : BOOL;
	bArm2VertStn12Regular_17 AT %MX26248.17 : BOOL;
	bArm2VertStn12Regular_18 AT %MX26248.18 : BOOL;
	bArm2VertStn12Regular_19 AT %MX26248.19 : BOOL;
	bArm2VertStn12Regular_20 AT %MX26248.20 : BOOL;
	bArm2VertStn12Regular_21 AT %MX26248.21 : BOOL;
	bArm2VertStn12Regular_22 AT %MX26248.22 : BOOL;
	bArm2VertStn12Regular_23 AT %MX26248.23 : BOOL;
	bArm2VertStn12Regular_24 AT %MX26248.24 : BOOL;
	bArm2VertStn12Regular_25 AT %MX26248.25 : BOOL;
	bArm2VertStn12Regular_26 AT %MX26248.26 : BOOL;
	bArm2VertStn12Regular_27 AT %MX26248.27 : BOOL;
	bArm2VertStn12Regular_28 AT %MX26248.28 : BOOL;
	bArm2VertStn12Regular_29 AT %MX26248.29 : BOOL;
	bArm2VertStn12Regular_30 AT %MX26248.30 : BOOL;
	bArm2VertStn12Regular_31 AT %MX26248.31 : BOOL;

(* xxxxxxxxxxxxxxxxxxxxxxxxxxxxxxxxxxxxxxx Vert xxxxxxxxxxxxxxxxxxxxxxxxxxxxxxxxxxxxxxx*)
(*========= Up AgiUp BOOL LINK with %MX26300-MX26399 =========*)

	bArm2VertStn1AglUp_00 AT %MX26304.0 : BOOL;
	bArm2VertStn1AglUp_01 AT %MX26304.1 : BOOL;
	bArm2VertStn1AglUp_02 AT %MX26304.2 : BOOL;
	bArm2VertStn1AglUp_03 AT %MX26304.3 : BOOL;
	bArm2VertStn1AglUp_04 AT %MX26304.4 : BOOL;
	bArm2VertStn1AglUp_05 AT %MX26304.5 : BOOL;
	bArm2VertStn1AglUp_06 AT %MX26304.6 : BOOL;
	bArm2VertStn1AglUp_07 AT %MX26304.7 : BOOL;
	bArm2VertStn1AglUp_08 AT %MX26304.8 : BOOL;
	bArm2VertStn1AglUp_09 AT %MX26304.9 : BOOL;
	bArm2VertStn1AglUp_10 AT %MX26304.10 : BOOL;
	bArm2VertStn1AglUp_11 AT %MX26304.11 : BOOL;
	bArm2VertStn1AglUp_12 AT %MX26304.12 : BOOL;
	bArm2VertStn1AglUp_13 AT %MX26304.13 : BOOL;
	bArm2VertStn1AglUp_14 AT %MX26304.14 : BOOL;
	bArm2VertStn1AglUp_15 AT %MX26304.15 : BOOL;
	bArm2VertStn1AglUp_16 AT %MX26304.16 : BOOL;
	bArm2VertStn1AglUp_17 AT %MX26304.17 : BOOL;
	bArm2VertStn1AglUp_18 AT %MX26304.18 : BOOL;
	bArm2VertStn1AglUp_19 AT %MX26304.19 : BOOL;
	bArm2VertStn1AglUp_20 AT %MX26304.20 : BOOL;
	bArm2VertStn1AglUp_21 AT %MX26304.21 : BOOL;
	bArm2VertStn1AglUp_22 AT %MX26304.22 : BOOL;
	bArm2VertStn1AglUp_23 AT %MX26304.23 : BOOL;
	bArm2VertStn1AglUp_24 AT %MX26304.24 : BOOL;
	bArm2VertStn1AglUp_25 AT %MX26304.25 : BOOL;
	bArm2VertStn1AglUp_26 AT %MX26304.26 : BOOL;
	bArm2VertStn1AglUp_27 AT %MX26304.27 : BOOL;
	bArm2VertStn1AglUp_28 AT %MX26304.28 : BOOL;
	bArm2VertStn1AglUp_29 AT %MX26304.29 : BOOL;
	bArm2VertStn1AglUp_30 AT %MX26304.30 : BOOL;
	bArm2VertStn1AglUp_31 AT %MX26304.31 : BOOL;

	bArm2VertStn2AglUp_00 AT %MX26308.0 : BOOL;
	bArm2VertStn2AglUp_01 AT %MX26308.1 : BOOL;
	bArm2VertStn2AglUp_02 AT %MX26308.2 : BOOL;
	bArm2VertStn2AglUp_03 AT %MX26308.3 : BOOL;
	bArm2VertStn2AglUp_04 AT %MX26308.4 : BOOL;
	bArm2VertStn2AglUp_05 AT %MX26308.5 : BOOL;
	bArm2VertStn2AglUp_06 AT %MX26308.6 : BOOL;
	bArm2VertStn2AglUp_07 AT %MX26308.7 : BOOL;
	bArm2VertStn2AglUp_08 AT %MX26308.8 : BOOL;
	bArm2VertStn2AglUp_09 AT %MX26308.9 : BOOL;
	bArm2VertStn2AglUp_10 AT %MX26308.10 : BOOL;
	bArm2VertStn2AglUp_11 AT %MX26308.11 : BOOL;
	bArm2VertStn2AglUp_12 AT %MX26308.12 : BOOL;
	bArm2VertStn2AglUp_13 AT %MX26308.13 : BOOL;
	bArm2VertStn2AglUp_14 AT %MX26308.14 : BOOL;
	bArm2VertStn2AglUp_15 AT %MX26308.15 : BOOL;
	bArm2VertStn2AglUp_16 AT %MX26308.16 : BOOL;
	bArm2VertStn2AglUp_17 AT %MX26308.17 : BOOL;
	bArm2VertStn2AglUp_18 AT %MX26308.18 : BOOL;
	bArm2VertStn2AglUp_19 AT %MX26308.19 : BOOL;
	bArm2VertStn2AglUp_20 AT %MX26308.20 : BOOL;
	bArm2VertStn2AglUp_21 AT %MX26308.21 : BOOL;
	bArm2VertStn2AglUp_22 AT %MX26308.22 : BOOL;
	bArm2VertStn2AglUp_23 AT %MX26308.23 : BOOL;
	bArm2VertStn2AglUp_24 AT %MX26308.24 : BOOL;
	bArm2VertStn2AglUp_25 AT %MX26308.25 : BOOL;
	bArm2VertStn2AglUp_26 AT %MX26308.26 : BOOL;
	bArm2VertStn2AglUp_27 AT %MX26308.27 : BOOL;
	bArm2VertStn2AglUp_28 AT %MX26308.28 : BOOL;
	bArm2VertStn2AglUp_29 AT %MX26308.29 : BOOL;
	bArm2VertStn2AglUp_30 AT %MX26308.30 : BOOL;
	bArm2VertStn2AglUp_31 AT %MX26308.31 : BOOL;

	bArm2VertStn3AglUp_00 AT %MX26312.0 : BOOL;
	bArm2VertStn3AglUp_01 AT %MX26312.1 : BOOL;
	bArm2VertStn3AglUp_02 AT %MX26312.2 : BOOL;
	bArm2VertStn3AglUp_03 AT %MX26312.3 : BOOL;
	bArm2VertStn3AglUp_04 AT %MX26312.4 : BOOL;
	bArm2VertStn3AglUp_05 AT %MX26312.5 : BOOL;
	bArm2VertStn3AglUp_06 AT %MX26312.6 : BOOL;
	bArm2VertStn3AglUp_07 AT %MX26312.7 : BOOL;
	bArm2VertStn3AglUp_08 AT %MX26312.8 : BOOL;
	bArm2VertStn3AglUp_09 AT %MX26312.9 : BOOL;
	bArm2VertStn3AglUp_10 AT %MX26312.10 : BOOL;
	bArm2VertStn3AglUp_11 AT %MX26312.11 : BOOL;
	bArm2VertStn3AglUp_12 AT %MX26312.12 : BOOL;
	bArm2VertStn3AglUp_13 AT %MX26312.13 : BOOL;
	bArm2VertStn3AglUp_14 AT %MX26312.14 : BOOL;
	bArm2VertStn3AglUp_15 AT %MX26312.15 : BOOL;
	bArm2VertStn3AglUp_16 AT %MX26312.16 : BOOL;
	bArm2VertStn3AglUp_17 AT %MX26312.17 : BOOL;
	bArm2VertStn3AglUp_18 AT %MX26312.18 : BOOL;
	bArm2VertStn3AglUp_19 AT %MX26312.19 : BOOL;
	bArm2VertStn3AglUp_20 AT %MX26312.20 : BOOL;
	bArm2VertStn3AglUp_21 AT %MX26312.21 : BOOL;
	bArm2VertStn3AglUp_22 AT %MX26312.22 : BOOL;
	bArm2VertStn3AglUp_23 AT %MX26312.23 : BOOL;
	bArm2VertStn3AglUp_24 AT %MX26312.24 : BOOL;
	bArm2VertStn3AglUp_25 AT %MX26312.25 : BOOL;
	bArm2VertStn3AglUp_26 AT %MX26312.26 : BOOL;
	bArm2VertStn3AglUp_27 AT %MX26312.27 : BOOL;
	bArm2VertStn3AglUp_28 AT %MX26312.28 : BOOL;
	bArm2VertStn3AglUp_29 AT %MX26312.29 : BOOL;
	bArm2VertStn3AglUp_30 AT %MX26312.30 : BOOL;
	bArm2VertStn3AglUp_31 AT %MX26312.31 : BOOL;

	bArm2VertStn4AglUp_00 AT %MX26316.0 : BOOL;
	bArm2VertStn4AglUp_01 AT %MX26316.1 : BOOL;
	bArm2VertStn4AglUp_02 AT %MX26316.2 : BOOL;
	bArm2VertStn4AglUp_03 AT %MX26316.3 : BOOL;
	bArm2VertStn4AglUp_04 AT %MX26316.4 : BOOL;
	bArm2VertStn4AglUp_05 AT %MX26316.5 : BOOL;
	bArm2VertStn4AglUp_06 AT %MX26316.6 : BOOL;
	bArm2VertStn4AglUp_07 AT %MX26316.7 : BOOL;
	bArm2VertStn4AglUp_08 AT %MX26316.8 : BOOL;
	bArm2VertStn4AglUp_09 AT %MX26316.9 : BOOL;
	bArm2VertStn4AglUp_10 AT %MX26316.10 : BOOL;
	bArm2VertStn4AglUp_11 AT %MX26316.11 : BOOL;
	bArm2VertStn4AglUp_12 AT %MX26316.12 : BOOL;
	bArm2VertStn4AglUp_13 AT %MX26316.13 : BOOL;
	bArm2VertStn4AglUp_14 AT %MX26316.14 : BOOL;
	bArm2VertStn4AglUp_15 AT %MX26316.15 : BOOL;
	bArm2VertStn4AglUp_16 AT %MX26316.16 : BOOL;
	bArm2VertStn4AglUp_17 AT %MX26316.17 : BOOL;
	bArm2VertStn4AglUp_18 AT %MX26316.18 : BOOL;
	bArm2VertStn4AglUp_19 AT %MX26316.19 : BOOL;
	bArm2VertStn4AglUp_20 AT %MX26316.20 : BOOL;
	bArm2VertStn4AglUp_21 AT %MX26316.21 : BOOL;
	bArm2VertStn4AglUp_22 AT %MX26316.22 : BOOL;
	bArm2VertStn4AglUp_23 AT %MX26316.23 : BOOL;
	bArm2VertStn4AglUp_24 AT %MX26316.24 : BOOL;
	bArm2VertStn4AglUp_25 AT %MX26316.25 : BOOL;
	bArm2VertStn4AglUp_26 AT %MX26316.26 : BOOL;
	bArm2VertStn4AglUp_27 AT %MX26316.27 : BOOL;
	bArm2VertStn4AglUp_28 AT %MX26316.28 : BOOL;
	bArm2VertStn4AglUp_29 AT %MX26316.29 : BOOL;
	bArm2VertStn4AglUp_30 AT %MX26316.30 : BOOL;
	bArm2VertStn4AglUp_31 AT %MX26316.31 : BOOL;

	bArm2VertStn5AglUp_00 AT %MX26320.0 : BOOL;
	bArm2VertStn5AglUp_01 AT %MX26320.1 : BOOL;
	bArm2VertStn5AglUp_02 AT %MX26320.2 : BOOL;
	bArm2VertStn5AglUp_03 AT %MX26320.3 : BOOL;
	bArm2VertStn5AglUp_04 AT %MX26320.4 : BOOL;
	bArm2VertStn5AglUp_05 AT %MX26320.5 : BOOL;
	bArm2VertStn5AglUp_06 AT %MX26320.6 : BOOL;
	bArm2VertStn5AglUp_07 AT %MX26320.7 : BOOL;
	bArm2VertStn5AglUp_08 AT %MX26320.8 : BOOL;
	bArm2VertStn5AglUp_09 AT %MX26320.9 : BOOL;
	bArm2VertStn5AglUp_10 AT %MX26320.10 : BOOL;
	bArm2VertStn5AglUp_11 AT %MX26320.11 : BOOL;
	bArm2VertStn5AglUp_12 AT %MX26320.12 : BOOL;
	bArm2VertStn5AglUp_13 AT %MX26320.13 : BOOL;
	bArm2VertStn5AglUp_14 AT %MX26320.14 : BOOL;
	bArm2VertStn5AglUp_15 AT %MX26320.15 : BOOL;
	bArm2VertStn5AglUp_16 AT %MX26320.16 : BOOL;
	bArm2VertStn5AglUp_17 AT %MX26320.17 : BOOL;
	bArm2VertStn5AglUp_18 AT %MX26320.18 : BOOL;
	bArm2VertStn5AglUp_19 AT %MX26320.19 : BOOL;
	bArm2VertStn5AglUp_20 AT %MX26320.20 : BOOL;
	bArm2VertStn5AglUp_21 AT %MX26320.21 : BOOL;
	bArm2VertStn5AglUp_22 AT %MX26320.22 : BOOL;
	bArm2VertStn5AglUp_23 AT %MX26320.23 : BOOL;
	bArm2VertStn5AglUp_24 AT %MX26320.24 : BOOL;
	bArm2VertStn5AglUp_25 AT %MX26320.25 : BOOL;
	bArm2VertStn5AglUp_26 AT %MX26320.26 : BOOL;
	bArm2VertStn5AglUp_27 AT %MX26320.27 : BOOL;
	bArm2VertStn5AglUp_28 AT %MX26320.28 : BOOL;
	bArm2VertStn5AglUp_29 AT %MX26320.29 : BOOL;
	bArm2VertStn5AglUp_30 AT %MX26320.30 : BOOL;
	bArm2VertStn5AglUp_31 AT %MX26320.31 : BOOL;

	bArm2VertStn6AglUp_00 AT %MX26324.0 : BOOL;
	bArm2VertStn6AglUp_01 AT %MX26324.1 : BOOL;
	bArm2VertStn6AglUp_02 AT %MX26324.2 : BOOL;
	bArm2VertStn6AglUp_03 AT %MX26324.3 : BOOL;
	bArm2VertStn6AglUp_04 AT %MX26324.4 : BOOL;
	bArm2VertStn6AglUp_05 AT %MX26324.5 : BOOL;
	bArm2VertStn6AglUp_06 AT %MX26324.6 : BOOL;
	bArm2VertStn6AglUp_07 AT %MX26324.7 : BOOL;
	bArm2VertStn6AglUp_08 AT %MX26324.8 : BOOL;
	bArm2VertStn6AglUp_09 AT %MX26324.9 : BOOL;
	bArm2VertStn6AglUp_10 AT %MX26324.10 : BOOL;
	bArm2VertStn6AglUp_11 AT %MX26324.11 : BOOL;
	bArm2VertStn6AglUp_12 AT %MX26324.12 : BOOL;
	bArm2VertStn6AglUp_13 AT %MX26324.13 : BOOL;
	bArm2VertStn6AglUp_14 AT %MX26324.14 : BOOL;
	bArm2VertStn6AglUp_15 AT %MX26324.15 : BOOL;
	bArm2VertStn6AglUp_16 AT %MX26324.16 : BOOL;
	bArm2VertStn6AglUp_17 AT %MX26324.17 : BOOL;
	bArm2VertStn6AglUp_18 AT %MX26324.18 : BOOL;
	bArm2VertStn6AglUp_19 AT %MX26324.19 : BOOL;
	bArm2VertStn6AglUp_20 AT %MX26324.20 : BOOL;
	bArm2VertStn6AglUp_21 AT %MX26324.21 : BOOL;
	bArm2VertStn6AglUp_22 AT %MX26324.22 : BOOL;
	bArm2VertStn6AglUp_23 AT %MX26324.23 : BOOL;
	bArm2VertStn6AglUp_24 AT %MX26324.24 : BOOL;
	bArm2VertStn6AglUp_25 AT %MX26324.25 : BOOL;
	bArm2VertStn6AglUp_26 AT %MX26324.26 : BOOL;
	bArm2VertStn6AglUp_27 AT %MX26324.27 : BOOL;
	bArm2VertStn6AglUp_28 AT %MX26324.28 : BOOL;
	bArm2VertStn6AglUp_29 AT %MX26324.29 : BOOL;
	bArm2VertStn6AglUp_30 AT %MX26324.30 : BOOL;
	bArm2VertStn6AglUp_31 AT %MX26324.31 : BOOL;

	bArm2VertStn7AglUp_00 AT %MX26328.0 : BOOL;
	bArm2VertStn7AglUp_01 AT %MX26328.1 : BOOL;
	bArm2VertStn7AglUp_02 AT %MX26328.2 : BOOL;
	bArm2VertStn7AglUp_03 AT %MX26328.3 : BOOL;
	bArm2VertStn7AglUp_04 AT %MX26328.4 : BOOL;
	bArm2VertStn7AglUp_05 AT %MX26328.5 : BOOL;
	bArm2VertStn7AglUp_06 AT %MX26328.6 : BOOL;
	bArm2VertStn7AglUp_07 AT %MX26328.7 : BOOL;
	bArm2VertStn7AglUp_08 AT %MX26328.8 : BOOL;
	bArm2VertStn7AglUp_09 AT %MX26328.9 : BOOL;
	bArm2VertStn7AglUp_10 AT %MX26328.10 : BOOL;
	bArm2VertStn7AglUp_11 AT %MX26328.11 : BOOL;
	bArm2VertStn7AglUp_12 AT %MX26328.12 : BOOL;
	bArm2VertStn7AglUp_13 AT %MX26328.13 : BOOL;
	bArm2VertStn7AglUp_14 AT %MX26328.14 : BOOL;
	bArm2VertStn7AglUp_15 AT %MX26328.15 : BOOL;
	bArm2VertStn7AglUp_16 AT %MX26328.16 : BOOL;
	bArm2VertStn7AglUp_17 AT %MX26328.17 : BOOL;
	bArm2VertStn7AglUp_18 AT %MX26328.18 : BOOL;
	bArm2VertStn7AglUp_19 AT %MX26328.19 : BOOL;
	bArm2VertStn7AglUp_20 AT %MX26328.20 : BOOL;
	bArm2VertStn7AglUp_21 AT %MX26328.21 : BOOL;
	bArm2VertStn7AglUp_22 AT %MX26328.22 : BOOL;
	bArm2VertStn7AglUp_23 AT %MX26328.23 : BOOL;
	bArm2VertStn7AglUp_24 AT %MX26328.24 : BOOL;
	bArm2VertStn7AglUp_25 AT %MX26328.25 : BOOL;
	bArm2VertStn7AglUp_26 AT %MX26328.26 : BOOL;
	bArm2VertStn7AglUp_27 AT %MX26328.27 : BOOL;
	bArm2VertStn7AglUp_28 AT %MX26328.28 : BOOL;
	bArm2VertStn7AglUp_29 AT %MX26328.29 : BOOL;
	bArm2VertStn7AglUp_30 AT %MX26328.30 : BOOL;
	bArm2VertStn7AglUp_31 AT %MX26328.31 : BOOL;

	bArm2VertStn8AglUp_00 AT %MX26332.0 : BOOL;
	bArm2VertStn8AglUp_01 AT %MX26332.1 : BOOL;
	bArm2VertStn8AglUp_02 AT %MX26332.2 : BOOL;
	bArm2VertStn8AglUp_03 AT %MX26332.3 : BOOL;
	bArm2VertStn8AglUp_04 AT %MX26332.4 : BOOL;
	bArm2VertStn8AglUp_05 AT %MX26332.5 : BOOL;
	bArm2VertStn8AglUp_06 AT %MX26332.6 : BOOL;
	bArm2VertStn8AglUp_07 AT %MX26332.7 : BOOL;
	bArm2VertStn8AglUp_08 AT %MX26332.8 : BOOL;
	bArm2VertStn8AglUp_09 AT %MX26332.9 : BOOL;
	bArm2VertStn8AglUp_10 AT %MX26332.10 : BOOL;
	bArm2VertStn8AglUp_11 AT %MX26332.11 : BOOL;
	bArm2VertStn8AglUp_12 AT %MX26332.12 : BOOL;
	bArm2VertStn8AglUp_13 AT %MX26332.13 : BOOL;
	bArm2VertStn8AglUp_14 AT %MX26332.14 : BOOL;
	bArm2VertStn8AglUp_15 AT %MX26332.15 : BOOL;
	bArm2VertStn8AglUp_16 AT %MX26332.16 : BOOL;
	bArm2VertStn8AglUp_17 AT %MX26332.17 : BOOL;
	bArm2VertStn8AglUp_18 AT %MX26332.18 : BOOL;
	bArm2VertStn8AglUp_19 AT %MX26332.19 : BOOL;
	bArm2VertStn8AglUp_20 AT %MX26332.20 : BOOL;
	bArm2VertStn8AglUp_21 AT %MX26332.21 : BOOL;
	bArm2VertStn8AglUp_22 AT %MX26332.22 : BOOL;
	bArm2VertStn8AglUp_23 AT %MX26332.23 : BOOL;
	bArm2VertStn8AglUp_24 AT %MX26332.24 : BOOL;
	bArm2VertStn8AglUp_25 AT %MX26332.25 : BOOL;
	bArm2VertStn8AglUp_26 AT %MX26332.26 : BOOL;
	bArm2VertStn8AglUp_27 AT %MX26332.27 : BOOL;
	bArm2VertStn8AglUp_28 AT %MX26332.28 : BOOL;
	bArm2VertStn8AglUp_29 AT %MX26332.29 : BOOL;
	bArm2VertStn8AglUp_30 AT %MX26332.30 : BOOL;
	bArm2VertStn8AglUp_31 AT %MX26332.31 : BOOL;

	bArm2VertStn9AglUp_00 AT %MX26336.0 : BOOL;
	bArm2VertStn9AglUp_01 AT %MX26336.1 : BOOL;
	bArm2VertStn9AglUp_02 AT %MX26336.2 : BOOL;
	bArm2VertStn9AglUp_03 AT %MX26336.3 : BOOL;
	bArm2VertStn9AglUp_04 AT %MX26336.4 : BOOL;
	bArm2VertStn9AglUp_05 AT %MX26336.5 : BOOL;
	bArm2VertStn9AglUp_06 AT %MX26336.6 : BOOL;
	bArm2VertStn9AglUp_07 AT %MX26336.7 : BOOL;
	bArm2VertStn9AglUp_08 AT %MX26336.8 : BOOL;
	bArm2VertStn9AglUp_09 AT %MX26336.9 : BOOL;
	bArm2VertStn9AglUp_10 AT %MX26336.10 : BOOL;
	bArm2VertStn9AglUp_11 AT %MX26336.11 : BOOL;
	bArm2VertStn9AglUp_12 AT %MX26336.12 : BOOL;
	bArm2VertStn9AglUp_13 AT %MX26336.13 : BOOL;
	bArm2VertStn9AglUp_14 AT %MX26336.14 : BOOL;
	bArm2VertStn9AglUp_15 AT %MX26336.15 : BOOL;
	bArm2VertStn9AglUp_16 AT %MX26336.16 : BOOL;
	bArm2VertStn9AglUp_17 AT %MX26336.17 : BOOL;
	bArm2VertStn9AglUp_18 AT %MX26336.18 : BOOL;
	bArm2VertStn9AglUp_19 AT %MX26336.19 : BOOL;
	bArm2VertStn9AglUp_20 AT %MX26336.20 : BOOL;
	bArm2VertStn9AglUp_21 AT %MX26336.21 : BOOL;
	bArm2VertStn9AglUp_22 AT %MX26336.22 : BOOL;
	bArm2VertStn9AglUp_23 AT %MX26336.23 : BOOL;
	bArm2VertStn9AglUp_24 AT %MX26336.24 : BOOL;
	bArm2VertStn9AglUp_25 AT %MX26336.25 : BOOL;
	bArm2VertStn9AglUp_26 AT %MX26336.26 : BOOL;
	bArm2VertStn9AglUp_27 AT %MX26336.27 : BOOL;
	bArm2VertStn9AglUp_28 AT %MX26336.28 : BOOL;
	bArm2VertStn9AglUp_29 AT %MX26336.29 : BOOL;
	bArm2VertStn9AglUp_30 AT %MX26336.30 : BOOL;
	bArm2VertStn9AglUp_31 AT %MX26336.31 : BOOL;

	bArm2VertStn10AglUp_00 AT %MX26340.0 : BOOL;
	bArm2VertStn10AglUp_01 AT %MX26340.1 : BOOL;
	bArm2VertStn10AglUp_02 AT %MX26340.2 : BOOL;
	bArm2VertStn10AglUp_03 AT %MX26340.3 : BOOL;
	bArm2VertStn10AglUp_04 AT %MX26340.4 : BOOL;
	bArm2VertStn10AglUp_05 AT %MX26340.5 : BOOL;
	bArm2VertStn10AglUp_06 AT %MX26340.6 : BOOL;
	bArm2VertStn10AglUp_07 AT %MX26340.7 : BOOL;
	bArm2VertStn10AglUp_08 AT %MX26340.8 : BOOL;
	bArm2VertStn10AglUp_09 AT %MX26340.9 : BOOL;
	bArm2VertStn10AglUp_10 AT %MX26340.10 : BOOL;
	bArm2VertStn10AglUp_11 AT %MX26340.11 : BOOL;
	bArm2VertStn10AglUp_12 AT %MX26340.12 : BOOL;
	bArm2VertStn10AglUp_13 AT %MX26340.13 : BOOL;
	bArm2VertStn10AglUp_14 AT %MX26340.14 : BOOL;
	bArm2VertStn10AglUp_15 AT %MX26340.15 : BOOL;
	bArm2VertStn10AglUp_16 AT %MX26340.16 : BOOL;
	bArm2VertStn10AglUp_17 AT %MX26340.17 : BOOL;
	bArm2VertStn10AglUp_18 AT %MX26340.18 : BOOL;
	bArm2VertStn10AglUp_19 AT %MX26340.19 : BOOL;
	bArm2VertStn10AglUp_20 AT %MX26340.20 : BOOL;
	bArm2VertStn10AglUp_21 AT %MX26340.21 : BOOL;
	bArm2VertStn10AglUp_22 AT %MX26340.22 : BOOL;
	bArm2VertStn10AglUp_23 AT %MX26340.23 : BOOL;
	bArm2VertStn10AglUp_24 AT %MX26340.24 : BOOL;
	bArm2VertStn10AglUp_25 AT %MX26340.25 : BOOL;
	bArm2VertStn10AglUp_26 AT %MX26340.26 : BOOL;
	bArm2VertStn10AglUp_27 AT %MX26340.27 : BOOL;
	bArm2VertStn10AglUp_28 AT %MX26340.28 : BOOL;
	bArm2VertStn10AglUp_29 AT %MX26340.29 : BOOL;
	bArm2VertStn10AglUp_30 AT %MX26340.30 : BOOL;
	bArm2VertStn10AglUp_31 AT %MX26340.31 : BOOL;

	bArm2VertStn11AglUp_00 AT %MX26344.0 : BOOL;
	bArm2VertStn11AglUp_01 AT %MX26344.1 : BOOL;
	bArm2VertStn11AglUp_02 AT %MX26344.2 : BOOL;
	bArm2VertStn11AglUp_03 AT %MX26344.3 : BOOL;
	bArm2VertStn11AglUp_04 AT %MX26344.4 : BOOL;
	bArm2VertStn11AglUp_05 AT %MX26344.5 : BOOL;
	bArm2VertStn11AglUp_06 AT %MX26344.6 : BOOL;
	bArm2VertStn11AglUp_07 AT %MX26344.7 : BOOL;
	bArm2VertStn11AglUp_08 AT %MX26344.8 : BOOL;
	bArm2VertStn11AglUp_09 AT %MX26344.9 : BOOL;
	bArm2VertStn11AglUp_10 AT %MX26344.10 : BOOL;
	bArm2VertStn11AglUp_11 AT %MX26344.11 : BOOL;
	bArm2VertStn11AglUp_12 AT %MX26344.12 : BOOL;
	bArm2VertStn11AglUp_13 AT %MX26344.13 : BOOL;
	bArm2VertStn11AglUp_14 AT %MX26344.14 : BOOL;
	bArm2VertStn11AglUp_15 AT %MX26344.15 : BOOL;
	bArm2VertStn11AglUp_16 AT %MX26344.16 : BOOL;
	bArm2VertStn11AglUp_17 AT %MX26344.17 : BOOL;
	bArm2VertStn11AglUp_18 AT %MX26344.18 : BOOL;
	bArm2VertStn11AglUp_19 AT %MX26344.19 : BOOL;
	bArm2VertStn11AglUp_20 AT %MX26344.20 : BOOL;
	bArm2VertStn11AglUp_21 AT %MX26344.21 : BOOL;
	bArm2VertStn11AglUp_22 AT %MX26344.22 : BOOL;
	bArm2VertStn11AglUp_23 AT %MX26344.23 : BOOL;
	bArm2VertStn11AglUp_24 AT %MX26344.24 : BOOL;
	bArm2VertStn11AglUp_25 AT %MX26344.25 : BOOL;
	bArm2VertStn11AglUp_26 AT %MX26344.26 : BOOL;
	bArm2VertStn11AglUp_27 AT %MX26344.27 : BOOL;
	bArm2VertStn11AglUp_28 AT %MX26344.28 : BOOL;
	bArm2VertStn11AglUp_29 AT %MX26344.29 : BOOL;
	bArm2VertStn11AglUp_30 AT %MX26344.30 : BOOL;
	bArm2VertStn11AglUp_31 AT %MX26344.31 : BOOL;

	bArm2VertStn12AglUp_00 AT %MX26348.0 : BOOL;
	bArm2VertStn12AglUp_01 AT %MX26348.1 : BOOL;
	bArm2VertStn12AglUp_02 AT %MX26348.2 : BOOL;
	bArm2VertStn12AglUp_03 AT %MX26348.3 : BOOL;
	bArm2VertStn12AglUp_04 AT %MX26348.4 : BOOL;
	bArm2VertStn12AglUp_05 AT %MX26348.5 : BOOL;
	bArm2VertStn12AglUp_06 AT %MX26348.6 : BOOL;
	bArm2VertStn12AglUp_07 AT %MX26348.7 : BOOL;
	bArm2VertStn12AglUp_08 AT %MX26348.8 : BOOL;
	bArm2VertStn12AglUp_09 AT %MX26348.9 : BOOL;
	bArm2VertStn12AglUp_10 AT %MX26348.10 : BOOL;
	bArm2VertStn12AglUp_11 AT %MX26348.11 : BOOL;
	bArm2VertStn12AglUp_12 AT %MX26348.12 : BOOL;
	bArm2VertStn12AglUp_13 AT %MX26348.13 : BOOL;
	bArm2VertStn12AglUp_14 AT %MX26348.14 : BOOL;
	bArm2VertStn12AglUp_15 AT %MX26348.15 : BOOL;
	bArm2VertStn12AglUp_16 AT %MX26348.16 : BOOL;
	bArm2VertStn12AglUp_17 AT %MX26348.17 : BOOL;
	bArm2VertStn12AglUp_18 AT %MX26348.18 : BOOL;
	bArm2VertStn12AglUp_19 AT %MX26348.19 : BOOL;
	bArm2VertStn12AglUp_20 AT %MX26348.20 : BOOL;
	bArm2VertStn12AglUp_21 AT %MX26348.21 : BOOL;
	bArm2VertStn12AglUp_22 AT %MX26348.22 : BOOL;
	bArm2VertStn12AglUp_23 AT %MX26348.23 : BOOL;
	bArm2VertStn12AglUp_24 AT %MX26348.24 : BOOL;
	bArm2VertStn12AglUp_25 AT %MX26348.25 : BOOL;
	bArm2VertStn12AglUp_26 AT %MX26348.26 : BOOL;
	bArm2VertStn12AglUp_27 AT %MX26348.27 : BOOL;
	bArm2VertStn12AglUp_28 AT %MX26348.28 : BOOL;
	bArm2VertStn12AglUp_29 AT %MX26348.29 : BOOL;
	bArm2VertStn12AglUp_30 AT %MX26348.30 : BOOL;
	bArm2VertStn12AglUp_31 AT %MX26348.31 : BOOL;

(* xxxxxxxxxxxxxxxxxxxxxxxxxxxxxxxxxxxxxxx Vert xxxxxxxxxxxxxxxxxxxxxxxxxxxxxxxxxxxxxxx*)
(*========= Down AgiDown BOOL LINK with %MX26400-MX26499 =========*)

	bArm2VertStn1AglDown_00 AT %MX26404.0 : BOOL;
	bArm2VertStn1AglDown_01 AT %MX26404.1 : BOOL;
	bArm2VertStn1AglDown_02 AT %MX26404.2 : BOOL;
	bArm2VertStn1AglDown_03 AT %MX26404.3 : BOOL;
	bArm2VertStn1AglDown_04 AT %MX26404.4 : BOOL;
	bArm2VertStn1AglDown_05 AT %MX26404.5 : BOOL;
	bArm2VertStn1AglDown_06 AT %MX26404.6 : BOOL;
	bArm2VertStn1AglDown_07 AT %MX26404.7 : BOOL;
	bArm2VertStn1AglDown_08 AT %MX26404.8 : BOOL;
	bArm2VertStn1AglDown_09 AT %MX26404.9 : BOOL;
	bArm2VertStn1AglDown_10 AT %MX26404.10 : BOOL;
	bArm2VertStn1AglDown_11 AT %MX26404.11 : BOOL;
	bArm2VertStn1AglDown_12 AT %MX26404.12 : BOOL;
	bArm2VertStn1AglDown_13 AT %MX26404.13 : BOOL;
	bArm2VertStn1AglDown_14 AT %MX26404.14 : BOOL;
	bArm2VertStn1AglDown_15 AT %MX26404.15 : BOOL;
	bArm2VertStn1AglDown_16 AT %MX26404.16 : BOOL;
	bArm2VertStn1AglDown_17 AT %MX26404.17 : BOOL;
	bArm2VertStn1AglDown_18 AT %MX26404.18 : BOOL;
	bArm2VertStn1AglDown_19 AT %MX26404.19 : BOOL;
	bArm2VertStn1AglDown_20 AT %MX26404.20 : BOOL;
	bArm2VertStn1AglDown_21 AT %MX26404.21 : BOOL;
	bArm2VertStn1AglDown_22 AT %MX26404.22 : BOOL;
	bArm2VertStn1AglDown_23 AT %MX26404.23 : BOOL;
	bArm2VertStn1AglDown_24 AT %MX26404.24 : BOOL;
	bArm2VertStn1AglDown_25 AT %MX26404.25 : BOOL;
	bArm2VertStn1AglDown_26 AT %MX26404.26 : BOOL;
	bArm2VertStn1AglDown_27 AT %MX26404.27 : BOOL;
	bArm2VertStn1AglDown_28 AT %MX26404.28 : BOOL;
	bArm2VertStn1AglDown_29 AT %MX26404.29 : BOOL;
	bArm2VertStn1AglDown_30 AT %MX26404.30 : BOOL;
	bArm2VertStn1AglDown_31 AT %MX26404.31 : BOOL;

	bArm2VertStn2AglDown_00 AT %MX26408.0 : BOOL;
	bArm2VertStn2AglDown_01 AT %MX26408.1 : BOOL;
	bArm2VertStn2AglDown_02 AT %MX26408.2 : BOOL;
	bArm2VertStn2AglDown_03 AT %MX26408.3 : BOOL;
	bArm2VertStn2AglDown_04 AT %MX26408.4 : BOOL;
	bArm2VertStn2AglDown_05 AT %MX26408.5 : BOOL;
	bArm2VertStn2AglDown_06 AT %MX26408.6 : BOOL;
	bArm2VertStn2AglDown_07 AT %MX26408.7 : BOOL;
	bArm2VertStn2AglDown_08 AT %MX26408.8 : BOOL;
	bArm2VertStn2AglDown_09 AT %MX26408.9 : BOOL;
	bArm2VertStn2AglDown_10 AT %MX26408.10 : BOOL;
	bArm2VertStn2AglDown_11 AT %MX26408.11 : BOOL;
	bArm2VertStn2AglDown_12 AT %MX26408.12 : BOOL;
	bArm2VertStn2AglDown_13 AT %MX26408.13 : BOOL;
	bArm2VertStn2AglDown_14 AT %MX26408.14 : BOOL;
	bArm2VertStn2AglDown_15 AT %MX26408.15 : BOOL;
	bArm2VertStn2AglDown_16 AT %MX26408.16 : BOOL;
	bArm2VertStn2AglDown_17 AT %MX26408.17 : BOOL;
	bArm2VertStn2AglDown_18 AT %MX26408.18 : BOOL;
	bArm2VertStn2AglDown_19 AT %MX26408.19 : BOOL;
	bArm2VertStn2AglDown_20 AT %MX26408.20 : BOOL;
	bArm2VertStn2AglDown_21 AT %MX26408.21 : BOOL;
	bArm2VertStn2AglDown_22 AT %MX26408.22 : BOOL;
	bArm2VertStn2AglDown_23 AT %MX26408.23 : BOOL;
	bArm2VertStn2AglDown_24 AT %MX26408.24 : BOOL;
	bArm2VertStn2AglDown_25 AT %MX26408.25 : BOOL;
	bArm2VertStn2AglDown_26 AT %MX26408.26 : BOOL;
	bArm2VertStn2AglDown_27 AT %MX26408.27 : BOOL;
	bArm2VertStn2AglDown_28 AT %MX26408.28 : BOOL;
	bArm2VertStn2AglDown_29 AT %MX26408.29 : BOOL;
	bArm2VertStn2AglDown_30 AT %MX26408.30 : BOOL;
	bArm2VertStn2AglDown_31 AT %MX26408.31 : BOOL;

	bArm2VertStn3AglDown_00 AT %MX26412.0 : BOOL;
	bArm2VertStn3AglDown_01 AT %MX26412.1 : BOOL;
	bArm2VertStn3AglDown_02 AT %MX26412.2 : BOOL;
	bArm2VertStn3AglDown_03 AT %MX26412.3 : BOOL;
	bArm2VertStn3AglDown_04 AT %MX26412.4 : BOOL;
	bArm2VertStn3AglDown_05 AT %MX26412.5 : BOOL;
	bArm2VertStn3AglDown_06 AT %MX26412.6 : BOOL;
	bArm2VertStn3AglDown_07 AT %MX26412.7 : BOOL;
	bArm2VertStn3AglDown_08 AT %MX26412.8 : BOOL;
	bArm2VertStn3AglDown_09 AT %MX26412.9 : BOOL;
	bArm2VertStn3AglDown_10 AT %MX26412.10 : BOOL;
	bArm2VertStn3AglDown_11 AT %MX26412.11 : BOOL;
	bArm2VertStn3AglDown_12 AT %MX26412.12 : BOOL;
	bArm2VertStn3AglDown_13 AT %MX26412.13 : BOOL;
	bArm2VertStn3AglDown_14 AT %MX26412.14 : BOOL;
	bArm2VertStn3AglDown_15 AT %MX26412.15 : BOOL;
	bArm2VertStn3AglDown_16 AT %MX26412.16 : BOOL;
	bArm2VertStn3AglDown_17 AT %MX26412.17 : BOOL;
	bArm2VertStn3AglDown_18 AT %MX26412.18 : BOOL;
	bArm2VertStn3AglDown_19 AT %MX26412.19 : BOOL;
	bArm2VertStn3AglDown_20 AT %MX26412.20 : BOOL;
	bArm2VertStn3AglDown_21 AT %MX26412.21 : BOOL;
	bArm2VertStn3AglDown_22 AT %MX26412.22 : BOOL;
	bArm2VertStn3AglDown_23 AT %MX26412.23 : BOOL;
	bArm2VertStn3AglDown_24 AT %MX26412.24 : BOOL;
	bArm2VertStn3AglDown_25 AT %MX26412.25 : BOOL;
	bArm2VertStn3AglDown_26 AT %MX26412.26 : BOOL;
	bArm2VertStn3AglDown_27 AT %MX26412.27 : BOOL;
	bArm2VertStn3AglDown_28 AT %MX26412.28 : BOOL;
	bArm2VertStn3AglDown_29 AT %MX26412.29 : BOOL;
	bArm2VertStn3AglDown_30 AT %MX26412.30 : BOOL;
	bArm2VertStn3AglDown_31 AT %MX26412.31 : BOOL;

	bArm2VertStn4AglDown_00 AT %MX26416.0 : BOOL;
	bArm2VertStn4AglDown_01 AT %MX26416.1 : BOOL;
	bArm2VertStn4AglDown_02 AT %MX26416.2 : BOOL;
	bArm2VertStn4AglDown_03 AT %MX26416.3 : BOOL;
	bArm2VertStn4AglDown_04 AT %MX26416.4 : BOOL;
	bArm2VertStn4AglDown_05 AT %MX26416.5 : BOOL;
	bArm2VertStn4AglDown_06 AT %MX26416.6 : BOOL;
	bArm2VertStn4AglDown_07 AT %MX26416.7 : BOOL;
	bArm2VertStn4AglDown_08 AT %MX26416.8 : BOOL;
	bArm2VertStn4AglDown_09 AT %MX26416.9 : BOOL;
	bArm2VertStn4AglDown_10 AT %MX26416.10 : BOOL;
	bArm2VertStn4AglDown_11 AT %MX26416.11 : BOOL;
	bArm2VertStn4AglDown_12 AT %MX26416.12 : BOOL;
	bArm2VertStn4AglDown_13 AT %MX26416.13 : BOOL;
	bArm2VertStn4AglDown_14 AT %MX26416.14 : BOOL;
	bArm2VertStn4AglDown_15 AT %MX26416.15 : BOOL;
	bArm2VertStn4AglDown_16 AT %MX26416.16 : BOOL;
	bArm2VertStn4AglDown_17 AT %MX26416.17 : BOOL;
	bArm2VertStn4AglDown_18 AT %MX26416.18 : BOOL;
	bArm2VertStn4AglDown_19 AT %MX26416.19 : BOOL;
	bArm2VertStn4AglDown_20 AT %MX26416.20 : BOOL;
	bArm2VertStn4AglDown_21 AT %MX26416.21 : BOOL;
	bArm2VertStn4AglDown_22 AT %MX26416.22 : BOOL;
	bArm2VertStn4AglDown_23 AT %MX26416.23 : BOOL;
	bArm2VertStn4AglDown_24 AT %MX26416.24 : BOOL;
	bArm2VertStn4AglDown_25 AT %MX26416.25 : BOOL;
	bArm2VertStn4AglDown_26 AT %MX26416.26 : BOOL;
	bArm2VertStn4AglDown_27 AT %MX26416.27 : BOOL;
	bArm2VertStn4AglDown_28 AT %MX26416.28 : BOOL;
	bArm2VertStn4AglDown_29 AT %MX26416.29 : BOOL;
	bArm2VertStn4AglDown_30 AT %MX26416.30 : BOOL;
	bArm2VertStn4AglDown_31 AT %MX26416.31 : BOOL;

	bArm2VertStn5AglDown_00 AT %MX26420.0 : BOOL;
	bArm2VertStn5AglDown_01 AT %MX26420.1 : BOOL;
	bArm2VertStn5AglDown_02 AT %MX26420.2 : BOOL;
	bArm2VertStn5AglDown_03 AT %MX26420.3 : BOOL;
	bArm2VertStn5AglDown_04 AT %MX26420.4 : BOOL;
	bArm2VertStn5AglDown_05 AT %MX26420.5 : BOOL;
	bArm2VertStn5AglDown_06 AT %MX26420.6 : BOOL;
	bArm2VertStn5AglDown_07 AT %MX26420.7 : BOOL;
	bArm2VertStn5AglDown_08 AT %MX26420.8 : BOOL;
	bArm2VertStn5AglDown_09 AT %MX26420.9 : BOOL;
	bArm2VertStn5AglDown_10 AT %MX26420.10 : BOOL;
	bArm2VertStn5AglDown_11 AT %MX26420.11 : BOOL;
	bArm2VertStn5AglDown_12 AT %MX26420.12 : BOOL;
	bArm2VertStn5AglDown_13 AT %MX26420.13 : BOOL;
	bArm2VertStn5AglDown_14 AT %MX26420.14 : BOOL;
	bArm2VertStn5AglDown_15 AT %MX26420.15 : BOOL;
	bArm2VertStn5AglDown_16 AT %MX26420.16 : BOOL;
	bArm2VertStn5AglDown_17 AT %MX26420.17 : BOOL;
	bArm2VertStn5AglDown_18 AT %MX26420.18 : BOOL;
	bArm2VertStn5AglDown_19 AT %MX26420.19 : BOOL;
	bArm2VertStn5AglDown_20 AT %MX26420.20 : BOOL;
	bArm2VertStn5AglDown_21 AT %MX26420.21 : BOOL;
	bArm2VertStn5AglDown_22 AT %MX26420.22 : BOOL;
	bArm2VertStn5AglDown_23 AT %MX26420.23 : BOOL;
	bArm2VertStn5AglDown_24 AT %MX26420.24 : BOOL;
	bArm2VertStn5AglDown_25 AT %MX26420.25 : BOOL;
	bArm2VertStn5AglDown_26 AT %MX26420.26 : BOOL;
	bArm2VertStn5AglDown_27 AT %MX26420.27 : BOOL;
	bArm2VertStn5AglDown_28 AT %MX26420.28 : BOOL;
	bArm2VertStn5AglDown_29 AT %MX26420.29 : BOOL;
	bArm2VertStn5AglDown_30 AT %MX26420.30 : BOOL;
	bArm2VertStn5AglDown_31 AT %MX26420.31 : BOOL;

	bArm2VertStn6AglDown_00 AT %MX26424.0 : BOOL;
	bArm2VertStn6AglDown_01 AT %MX26424.1 : BOOL;
	bArm2VertStn6AglDown_02 AT %MX26424.2 : BOOL;
	bArm2VertStn6AglDown_03 AT %MX26424.3 : BOOL;
	bArm2VertStn6AglDown_04 AT %MX26424.4 : BOOL;
	bArm2VertStn6AglDown_05 AT %MX26424.5 : BOOL;
	bArm2VertStn6AglDown_06 AT %MX26424.6 : BOOL;
	bArm2VertStn6AglDown_07 AT %MX26424.7 : BOOL;
	bArm2VertStn6AglDown_08 AT %MX26424.8 : BOOL;
	bArm2VertStn6AglDown_09 AT %MX26424.9 : BOOL;
	bArm2VertStn6AglDown_10 AT %MX26424.10 : BOOL;
	bArm2VertStn6AglDown_11 AT %MX26424.11 : BOOL;
	bArm2VertStn6AglDown_12 AT %MX26424.12 : BOOL;
	bArm2VertStn6AglDown_13 AT %MX26424.13 : BOOL;
	bArm2VertStn6AglDown_14 AT %MX26424.14 : BOOL;
	bArm2VertStn6AglDown_15 AT %MX26424.15 : BOOL;
	bArm2VertStn6AglDown_16 AT %MX26424.16 : BOOL;
	bArm2VertStn6AglDown_17 AT %MX26424.17 : BOOL;
	bArm2VertStn6AglDown_18 AT %MX26424.18 : BOOL;
	bArm2VertStn6AglDown_19 AT %MX26424.19 : BOOL;
	bArm2VertStn6AglDown_20 AT %MX26424.20 : BOOL;
	bArm2VertStn6AglDown_21 AT %MX26424.21 : BOOL;
	bArm2VertStn6AglDown_22 AT %MX26424.22 : BOOL;
	bArm2VertStn6AglDown_23 AT %MX26424.23 : BOOL;
	bArm2VertStn6AglDown_24 AT %MX26424.24 : BOOL;
	bArm2VertStn6AglDown_25 AT %MX26424.25 : BOOL;
	bArm2VertStn6AglDown_26 AT %MX26424.26 : BOOL;
	bArm2VertStn6AglDown_27 AT %MX26424.27 : BOOL;
	bArm2VertStn6AglDown_28 AT %MX26424.28 : BOOL;
	bArm2VertStn6AglDown_29 AT %MX26424.29 : BOOL;
	bArm2VertStn6AglDown_30 AT %MX26424.30 : BOOL;
	bArm2VertStn6AglDown_31 AT %MX26424.31 : BOOL;

	bArm2VertStn7AglDown_00 AT %MX26428.0 : BOOL;
	bArm2VertStn7AglDown_01 AT %MX26428.1 : BOOL;
	bArm2VertStn7AglDown_02 AT %MX26428.2 : BOOL;
	bArm2VertStn7AglDown_03 AT %MX26428.3 : BOOL;
	bArm2VertStn7AglDown_04 AT %MX26428.4 : BOOL;
	bArm2VertStn7AglDown_05 AT %MX26428.5 : BOOL;
	bArm2VertStn7AglDown_06 AT %MX26428.6 : BOOL;
	bArm2VertStn7AglDown_07 AT %MX26428.7 : BOOL;
	bArm2VertStn7AglDown_08 AT %MX26428.8 : BOOL;
	bArm2VertStn7AglDown_09 AT %MX26428.9 : BOOL;
	bArm2VertStn7AglDown_10 AT %MX26428.10 : BOOL;
	bArm2VertStn7AglDown_11 AT %MX26428.11 : BOOL;
	bArm2VertStn7AglDown_12 AT %MX26428.12 : BOOL;
	bArm2VertStn7AglDown_13 AT %MX26428.13 : BOOL;
	bArm2VertStn7AglDown_14 AT %MX26428.14 : BOOL;
	bArm2VertStn7AglDown_15 AT %MX26428.15 : BOOL;
	bArm2VertStn7AglDown_16 AT %MX26428.16 : BOOL;
	bArm2VertStn7AglDown_17 AT %MX26428.17 : BOOL;
	bArm2VertStn7AglDown_18 AT %MX26428.18 : BOOL;
	bArm2VertStn7AglDown_19 AT %MX26428.19 : BOOL;
	bArm2VertStn7AglDown_20 AT %MX26428.20 : BOOL;
	bArm2VertStn7AglDown_21 AT %MX26428.21 : BOOL;
	bArm2VertStn7AglDown_22 AT %MX26428.22 : BOOL;
	bArm2VertStn7AglDown_23 AT %MX26428.23 : BOOL;
	bArm2VertStn7AglDown_24 AT %MX26428.24 : BOOL;
	bArm2VertStn7AglDown_25 AT %MX26428.25 : BOOL;
	bArm2VertStn7AglDown_26 AT %MX26428.26 : BOOL;
	bArm2VertStn7AglDown_27 AT %MX26428.27 : BOOL;
	bArm2VertStn7AglDown_28 AT %MX26428.28 : BOOL;
	bArm2VertStn7AglDown_29 AT %MX26428.29 : BOOL;
	bArm2VertStn7AglDown_30 AT %MX26428.30 : BOOL;
	bArm2VertStn7AglDown_31 AT %MX26428.31 : BOOL;

	bArm2VertStn8AglDown_00 AT %MX26432.0 : BOOL;
	bArm2VertStn8AglDown_01 AT %MX26432.1 : BOOL;
	bArm2VertStn8AglDown_02 AT %MX26432.2 : BOOL;
	bArm2VertStn8AglDown_03 AT %MX26432.3 : BOOL;
	bArm2VertStn8AglDown_04 AT %MX26432.4 : BOOL;
	bArm2VertStn8AglDown_05 AT %MX26432.5 : BOOL;
	bArm2VertStn8AglDown_06 AT %MX26432.6 : BOOL;
	bArm2VertStn8AglDown_07 AT %MX26432.7 : BOOL;
	bArm2VertStn8AglDown_08 AT %MX26432.8 : BOOL;
	bArm2VertStn8AglDown_09 AT %MX26432.9 : BOOL;
	bArm2VertStn8AglDown_10 AT %MX26432.10 : BOOL;
	bArm2VertStn8AglDown_11 AT %MX26432.11 : BOOL;
	bArm2VertStn8AglDown_12 AT %MX26432.12 : BOOL;
	bArm2VertStn8AglDown_13 AT %MX26432.13 : BOOL;
	bArm2VertStn8AglDown_14 AT %MX26432.14 : BOOL;
	bArm2VertStn8AglDown_15 AT %MX26432.15 : BOOL;
	bArm2VertStn8AglDown_16 AT %MX26432.16 : BOOL;
	bArm2VertStn8AglDown_17 AT %MX26432.17 : BOOL;
	bArm2VertStn8AglDown_18 AT %MX26432.18 : BOOL;
	bArm2VertStn8AglDown_19 AT %MX26432.19 : BOOL;
	bArm2VertStn8AglDown_20 AT %MX26432.20 : BOOL;
	bArm2VertStn8AglDown_21 AT %MX26432.21 : BOOL;
	bArm2VertStn8AglDown_22 AT %MX26432.22 : BOOL;
	bArm2VertStn8AglDown_23 AT %MX26432.23 : BOOL;
	bArm2VertStn8AglDown_24 AT %MX26432.24 : BOOL;
	bArm2VertStn8AglDown_25 AT %MX26432.25 : BOOL;
	bArm2VertStn8AglDown_26 AT %MX26432.26 : BOOL;
	bArm2VertStn8AglDown_27 AT %MX26432.27 : BOOL;
	bArm2VertStn8AglDown_28 AT %MX26432.28 : BOOL;
	bArm2VertStn8AglDown_29 AT %MX26432.29 : BOOL;
	bArm2VertStn8AglDown_30 AT %MX26432.30 : BOOL;
	bArm2VertStn8AglDown_31 AT %MX26432.31 : BOOL;

	bArm2VertStn9AglDown_00 AT %MX26436.0 : BOOL;
	bArm2VertStn9AglDown_01 AT %MX26436.1 : BOOL;
	bArm2VertStn9AglDown_02 AT %MX26436.2 : BOOL;
	bArm2VertStn9AglDown_03 AT %MX26436.3 : BOOL;
	bArm2VertStn9AglDown_04 AT %MX26436.4 : BOOL;
	bArm2VertStn9AglDown_05 AT %MX26436.5 : BOOL;
	bArm2VertStn9AglDown_06 AT %MX26436.6 : BOOL;
	bArm2VertStn9AglDown_07 AT %MX26436.7 : BOOL;
	bArm2VertStn9AglDown_08 AT %MX26436.8 : BOOL;
	bArm2VertStn9AglDown_09 AT %MX26436.9 : BOOL;
	bArm2VertStn9AglDown_10 AT %MX26436.10 : BOOL;
	bArm2VertStn9AglDown_11 AT %MX26436.11 : BOOL;
	bArm2VertStn9AglDown_12 AT %MX26436.12 : BOOL;
	bArm2VertStn9AglDown_13 AT %MX26436.13 : BOOL;
	bArm2VertStn9AglDown_14 AT %MX26436.14 : BOOL;
	bArm2VertStn9AglDown_15 AT %MX26436.15 : BOOL;
	bArm2VertStn9AglDown_16 AT %MX26436.16 : BOOL;
	bArm2VertStn9AglDown_17 AT %MX26436.17 : BOOL;
	bArm2VertStn9AglDown_18 AT %MX26436.18 : BOOL;
	bArm2VertStn9AglDown_19 AT %MX26436.19 : BOOL;
	bArm2VertStn9AglDown_20 AT %MX26436.20 : BOOL;
	bArm2VertStn9AglDown_21 AT %MX26436.21 : BOOL;
	bArm2VertStn9AglDown_22 AT %MX26436.22 : BOOL;
	bArm2VertStn9AglDown_23 AT %MX26436.23 : BOOL;
	bArm2VertStn9AglDown_24 AT %MX26436.24 : BOOL;
	bArm2VertStn9AglDown_25 AT %MX26436.25 : BOOL;
	bArm2VertStn9AglDown_26 AT %MX26436.26 : BOOL;
	bArm2VertStn9AglDown_27 AT %MX26436.27 : BOOL;
	bArm2VertStn9AglDown_28 AT %MX26436.28 : BOOL;
	bArm2VertStn9AglDown_29 AT %MX26436.29 : BOOL;
	bArm2VertStn9AglDown_30 AT %MX26436.30 : BOOL;
	bArm2VertStn9AglDown_31 AT %MX26436.31 : BOOL;

	bArm2VertStn10AglDown_00 AT %MX26440.0 : BOOL;
	bArm2VertStn10AglDown_01 AT %MX26440.1 : BOOL;
	bArm2VertStn10AglDown_02 AT %MX26440.2 : BOOL;
	bArm2VertStn10AglDown_03 AT %MX26440.3 : BOOL;
	bArm2VertStn10AglDown_04 AT %MX26440.4 : BOOL;
	bArm2VertStn10AglDown_05 AT %MX26440.5 : BOOL;
	bArm2VertStn10AglDown_06 AT %MX26440.6 : BOOL;
	bArm2VertStn10AglDown_07 AT %MX26440.7 : BOOL;
	bArm2VertStn10AglDown_08 AT %MX26440.8 : BOOL;
	bArm2VertStn10AglDown_09 AT %MX26440.9 : BOOL;
	bArm2VertStn10AglDown_10 AT %MX26440.10 : BOOL;
	bArm2VertStn10AglDown_11 AT %MX26440.11 : BOOL;
	bArm2VertStn10AglDown_12 AT %MX26440.12 : BOOL;
	bArm2VertStn10AglDown_13 AT %MX26440.13 : BOOL;
	bArm2VertStn10AglDown_14 AT %MX26440.14 : BOOL;
	bArm2VertStn10AglDown_15 AT %MX26440.15 : BOOL;
	bArm2VertStn10AglDown_16 AT %MX26440.16 : BOOL;
	bArm2VertStn10AglDown_17 AT %MX26440.17 : BOOL;
	bArm2VertStn10AglDown_18 AT %MX26440.18 : BOOL;
	bArm2VertStn10AglDown_19 AT %MX26440.19 : BOOL;
	bArm2VertStn10AglDown_20 AT %MX26440.20 : BOOL;
	bArm2VertStn10AglDown_21 AT %MX26440.21 : BOOL;
	bArm2VertStn10AglDown_22 AT %MX26440.22 : BOOL;
	bArm2VertStn10AglDown_23 AT %MX26440.23 : BOOL;
	bArm2VertStn10AglDown_24 AT %MX26440.24 : BOOL;
	bArm2VertStn10AglDown_25 AT %MX26440.25 : BOOL;
	bArm2VertStn10AglDown_26 AT %MX26440.26 : BOOL;
	bArm2VertStn10AglDown_27 AT %MX26440.27 : BOOL;
	bArm2VertStn10AglDown_28 AT %MX26440.28 : BOOL;
	bArm2VertStn10AglDown_29 AT %MX26440.29 : BOOL;
	bArm2VertStn10AglDown_30 AT %MX26440.30 : BOOL;
	bArm2VertStn10AglDown_31 AT %MX26440.31 : BOOL;

	bArm2VertStn11AglDown_00 AT %MX26444.0 : BOOL;
	bArm2VertStn11AglDown_01 AT %MX26444.1 : BOOL;
	bArm2VertStn11AglDown_02 AT %MX26444.2 : BOOL;
	bArm2VertStn11AglDown_03 AT %MX26444.3 : BOOL;
	bArm2VertStn11AglDown_04 AT %MX26444.4 : BOOL;
	bArm2VertStn11AglDown_05 AT %MX26444.5 : BOOL;
	bArm2VertStn11AglDown_06 AT %MX26444.6 : BOOL;
	bArm2VertStn11AglDown_07 AT %MX26444.7 : BOOL;
	bArm2VertStn11AglDown_08 AT %MX26444.8 : BOOL;
	bArm2VertStn11AglDown_09 AT %MX26444.9 : BOOL;
	bArm2VertStn11AglDown_10 AT %MX26444.10 : BOOL;
	bArm2VertStn11AglDown_11 AT %MX26444.11 : BOOL;
	bArm2VertStn11AglDown_12 AT %MX26444.12 : BOOL;
	bArm2VertStn11AglDown_13 AT %MX26444.13 : BOOL;
	bArm2VertStn11AglDown_14 AT %MX26444.14 : BOOL;
	bArm2VertStn11AglDown_15 AT %MX26444.15 : BOOL;
	bArm2VertStn11AglDown_16 AT %MX26444.16 : BOOL;
	bArm2VertStn11AglDown_17 AT %MX26444.17 : BOOL;
	bArm2VertStn11AglDown_18 AT %MX26444.18 : BOOL;
	bArm2VertStn11AglDown_19 AT %MX26444.19 : BOOL;
	bArm2VertStn11AglDown_20 AT %MX26444.20 : BOOL;
	bArm2VertStn11AglDown_21 AT %MX26444.21 : BOOL;
	bArm2VertStn11AglDown_22 AT %MX26444.22 : BOOL;
	bArm2VertStn11AglDown_23 AT %MX26444.23 : BOOL;
	bArm2VertStn11AglDown_24 AT %MX26444.24 : BOOL;
	bArm2VertStn11AglDown_25 AT %MX26444.25 : BOOL;
	bArm2VertStn11AglDown_26 AT %MX26444.26 : BOOL;
	bArm2VertStn11AglDown_27 AT %MX26444.27 : BOOL;
	bArm2VertStn11AglDown_28 AT %MX26444.28 : BOOL;
	bArm2VertStn11AglDown_29 AT %MX26444.29 : BOOL;
	bArm2VertStn11AglDown_30 AT %MX26444.30 : BOOL;
	bArm2VertStn11AglDown_31 AT %MX26444.31 : BOOL;

	bArm2VertStn12AglDown_00 AT %MX26448.0 : BOOL;
	bArm2VertStn12AglDown_01 AT %MX26448.1 : BOOL;
	bArm2VertStn12AglDown_02 AT %MX26448.2 : BOOL;
	bArm2VertStn12AglDown_03 AT %MX26448.3 : BOOL;
	bArm2VertStn12AglDown_04 AT %MX26448.4 : BOOL;
	bArm2VertStn12AglDown_05 AT %MX26448.5 : BOOL;
	bArm2VertStn12AglDown_06 AT %MX26448.6 : BOOL;
	bArm2VertStn12AglDown_07 AT %MX26448.7 : BOOL;
	bArm2VertStn12AglDown_08 AT %MX26448.8 : BOOL;
	bArm2VertStn12AglDown_09 AT %MX26448.9 : BOOL;
	bArm2VertStn12AglDown_10 AT %MX26448.10 : BOOL;
	bArm2VertStn12AglDown_11 AT %MX26448.11 : BOOL;
	bArm2VertStn12AglDown_12 AT %MX26448.12 : BOOL;
	bArm2VertStn12AglDown_13 AT %MX26448.13 : BOOL;
	bArm2VertStn12AglDown_14 AT %MX26448.14 : BOOL;
	bArm2VertStn12AglDown_15 AT %MX26448.15 : BOOL;
	bArm2VertStn12AglDown_16 AT %MX26448.16 : BOOL;
	bArm2VertStn12AglDown_17 AT %MX26448.17 : BOOL;
	bArm2VertStn12AglDown_18 AT %MX26448.18 : BOOL;
	bArm2VertStn12AglDown_19 AT %MX26448.19 : BOOL;
	bArm2VertStn12AglDown_20 AT %MX26448.20 : BOOL;
	bArm2VertStn12AglDown_21 AT %MX26448.21 : BOOL;
	bArm2VertStn12AglDown_22 AT %MX26448.22 : BOOL;
	bArm2VertStn12AglDown_23 AT %MX26448.23 : BOOL;
	bArm2VertStn12AglDown_24 AT %MX26448.24 : BOOL;
	bArm2VertStn12AglDown_25 AT %MX26448.25 : BOOL;
	bArm2VertStn12AglDown_26 AT %MX26448.26 : BOOL;
	bArm2VertStn12AglDown_27 AT %MX26448.27 : BOOL;
	bArm2VertStn12AglDown_28 AT %MX26448.28 : BOOL;
	bArm2VertStn12AglDown_29 AT %MX26448.29 : BOOL;
	bArm2VertStn12AglDown_30 AT %MX26448.30 : BOOL;
	bArm2VertStn12AglDown_31 AT %MX26448.31 : BOOL;


(* xxxxxxxxxxxxxxxxxxxxxxxxxxxxxxxxxxxxxxx Vert xxxxxxxxxxxxxxxxxxxxxxxxxxxxxxxxxxxxxxx*)
(*========= Down BOOL LINK with %MX26500-MX26599 =========*)

	bArm2VertLD1Down_00 AT %MX26552.0 : BOOL;
	bArm2VertLD1Down_01 AT %MX26552.1 : BOOL;
	bArm2VertLD1Down_02 AT %MX26552.2 : BOOL;
	bArm2VertLD1Down_03 AT %MX26552.3 : BOOL;
	bArm2VertLD1Down_04 AT %MX26552.4 : BOOL;
	bArm2VertLD1Down_05 AT %MX26552.5 : BOOL;
	bArm2VertLD1Down_06 AT %MX26552.6 : BOOL;
	bArm2VertLD1Down_07 AT %MX26552.7 : BOOL;
	bArm2VertLD1Down_08 AT %MX26552.8 : BOOL;
	bArm2VertLD1Down_09 AT %MX26552.9 : BOOL;
	bArm2VertLD1Down_10 AT %MX26552.10 : BOOL;
	bArm2VertLD1Down_11 AT %MX26552.11 : BOOL;
	bArm2VertLD1Down_12 AT %MX26552.12 : BOOL;
	bArm2VertLD1Down_13 AT %MX26552.13 : BOOL;
	bArm2VertLD1Down_14 AT %MX26552.14 : BOOL;
	bArm2VertLD1Down_15 AT %MX26552.15 : BOOL;
	bArm2VertLD1Down_16 AT %MX26552.16 : BOOL;
	bArm2VertLD1Down_17 AT %MX26552.17 : BOOL;
	bArm2VertLD1Down_18 AT %MX26552.18 : BOOL;
	bArm2VertLD1Down_19 AT %MX26552.19 : BOOL;
	bArm2VertLD1Down_20 AT %MX26552.20 : BOOL;
	bArm2VertLD1Down_21 AT %MX26552.21 : BOOL;
	bArm2VertLD1Down_22 AT %MX26552.22 : BOOL;
	bArm2VertLD1Down_23 AT %MX26552.23 : BOOL;
	bArm2VertLD1Down_24 AT %MX26552.24 : BOOL;
	bArm2VertLD1Down_25 AT %MX26552.25 : BOOL;
	bArm2VertLD1Down_26 AT %MX26552.26 : BOOL;
	bArm2VertLD1Down_27 AT %MX26552.27 : BOOL;
	bArm2VertLD1Down_28 AT %MX26552.28 : BOOL;
	bArm2VertLD1Down_29 AT %MX26552.29 : BOOL;
	bArm2VertLD1Down_30 AT %MX26552.30 : BOOL;
	bArm2VertLD1Down_31 AT %MX26552.31 : BOOL;

	bArm2VertULD1Down_00 AT %MX26556.0 : BOOL;
	bArm2VertULD1Down_01 AT %MX26556.1 : BOOL;
	bArm2VertULD1Down_02 AT %MX26556.2 : BOOL;
	bArm2VertULD1Down_03 AT %MX26556.3 : BOOL;
	bArm2VertULD1Down_04 AT %MX26556.4 : BOOL;
	bArm2VertULD1Down_05 AT %MX26556.5 : BOOL;
	bArm2VertULD1Down_06 AT %MX26556.6 : BOOL;
	bArm2VertULD1Down_07 AT %MX26556.7 : BOOL;
	bArm2VertULD1Down_08 AT %MX26556.8 : BOOL;
	bArm2VertULD1Down_09 AT %MX26556.9 : BOOL;
	bArm2VertULD1Down_10 AT %MX26556.10 : BOOL;
	bArm2VertULD1Down_11 AT %MX26556.11 : BOOL;
	bArm2VertULD1Down_12 AT %MX26556.12 : BOOL;
	bArm2VertULD1Down_13 AT %MX26556.13 : BOOL;
	bArm2VertULD1Down_14 AT %MX26556.14 : BOOL;
	bArm2VertULD1Down_15 AT %MX26556.15 : BOOL;
	bArm2VertULD1Down_16 AT %MX26556.16 : BOOL;
	bArm2VertULD1Down_17 AT %MX26556.17 : BOOL;
	bArm2VertULD1Down_18 AT %MX26556.18 : BOOL;
	bArm2VertULD1Down_19 AT %MX26556.19 : BOOL;
	bArm2VertULD1Down_20 AT %MX26556.20 : BOOL;
	bArm2VertULD1Down_21 AT %MX26556.21 : BOOL;
	bArm2VertULD1Down_22 AT %MX26556.22 : BOOL;
	bArm2VertULD1Down_23 AT %MX26556.23 : BOOL;
	bArm2VertULD1Down_24 AT %MX26556.24 : BOOL;
	bArm2VertULD1Down_25 AT %MX26556.25 : BOOL;
	bArm2VertULD1Down_26 AT %MX26556.26 : BOOL;
	bArm2VertULD1Down_27 AT %MX26556.27 : BOOL;
	bArm2VertULD1Down_28 AT %MX26556.28 : BOOL;
	bArm2VertULD1Down_29 AT %MX26556.29 : BOOL;
	bArm2VertULD1Down_30 AT %MX26556.30 : BOOL;
	bArm2VertULD1Down_31 AT %MX26556.31 : BOOL;

	bArm2VertStn1Down_00 AT %MX26504.0 : BOOL;
	bArm2VertStn1Down_01 AT %MX26504.1 : BOOL;
	bArm2VertStn1Down_02 AT %MX26504.2 : BOOL;
	bArm2VertStn1Down_03 AT %MX26504.3 : BOOL;
	bArm2VertStn1Down_04 AT %MX26504.4 : BOOL;
	bArm2VertStn1Down_05 AT %MX26504.5 : BOOL;
	bArm2VertStn1Down_06 AT %MX26504.6 : BOOL;
	bArm2VertStn1Down_07 AT %MX26504.7 : BOOL;
	bArm2VertStn1Down_08 AT %MX26504.8 : BOOL;
	bArm2VertStn1Down_09 AT %MX26504.9 : BOOL;
	bArm2VertStn1Down_10 AT %MX26504.10 : BOOL;
	bArm2VertStn1Down_11 AT %MX26504.11 : BOOL;
	bArm2VertStn1Down_12 AT %MX26504.12 : BOOL;
	bArm2VertStn1Down_13 AT %MX26504.13 : BOOL;
	bArm2VertStn1Down_14 AT %MX26504.14 : BOOL;
	bArm2VertStn1Down_15 AT %MX26504.15 : BOOL;
	bArm2VertStn1Down_16 AT %MX26504.16 : BOOL;
	bArm2VertStn1Down_17 AT %MX26504.17 : BOOL;
	bArm2VertStn1Down_18 AT %MX26504.18 : BOOL;
	bArm2VertStn1Down_19 AT %MX26504.19 : BOOL;
	bArm2VertStn1Down_20 AT %MX26504.20 : BOOL;
	bArm2VertStn1Down_21 AT %MX26504.21 : BOOL;
	bArm2VertStn1Down_22 AT %MX26504.22 : BOOL;
	bArm2VertStn1Down_23 AT %MX26504.23 : BOOL;
	bArm2VertStn1Down_24 AT %MX26504.24 : BOOL;
	bArm2VertStn1Down_25 AT %MX26504.25 : BOOL;
	bArm2VertStn1Down_26 AT %MX26504.26 : BOOL;
	bArm2VertStn1Down_27 AT %MX26504.27 : BOOL;
	bArm2VertStn1Down_28 AT %MX26504.28 : BOOL;
	bArm2VertStn1Down_29 AT %MX26504.29 : BOOL;
	bArm2VertStn1Down_30 AT %MX26504.30 : BOOL;
	bArm2VertStn1Down_31 AT %MX26504.31 : BOOL;

	bArm2VertStn2Down_00 AT %MX26508.0 : BOOL;
	bArm2VertStn2Down_01 AT %MX26508.1 : BOOL;
	bArm2VertStn2Down_02 AT %MX26508.2 : BOOL;
	bArm2VertStn2Down_03 AT %MX26508.3 : BOOL;
	bArm2VertStn2Down_04 AT %MX26508.4 : BOOL;
	bArm2VertStn2Down_05 AT %MX26508.5 : BOOL;
	bArm2VertStn2Down_06 AT %MX26508.6 : BOOL;
	bArm2VertStn2Down_07 AT %MX26508.7 : BOOL;
	bArm2VertStn2Down_08 AT %MX26508.8 : BOOL;
	bArm2VertStn2Down_09 AT %MX26508.9 : BOOL;
	bArm2VertStn2Down_10 AT %MX26508.10 : BOOL;
	bArm2VertStn2Down_11 AT %MX26508.11 : BOOL;
	bArm2VertStn2Down_12 AT %MX26508.12 : BOOL;
	bArm2VertStn2Down_13 AT %MX26508.13 : BOOL;
	bArm2VertStn2Down_14 AT %MX26508.14 : BOOL;
	bArm2VertStn2Down_15 AT %MX26508.15 : BOOL;
	bArm2VertStn2Down_16 AT %MX26508.16 : BOOL;
	bArm2VertStn2Down_17 AT %MX26508.17 : BOOL;
	bArm2VertStn2Down_18 AT %MX26508.18 : BOOL;
	bArm2VertStn2Down_19 AT %MX26508.19 : BOOL;
	bArm2VertStn2Down_20 AT %MX26508.20 : BOOL;
	bArm2VertStn2Down_21 AT %MX26508.21 : BOOL;
	bArm2VertStn2Down_22 AT %MX26508.22 : BOOL;
	bArm2VertStn2Down_23 AT %MX26508.23 : BOOL;
	bArm2VertStn2Down_24 AT %MX26508.24 : BOOL;
	bArm2VertStn2Down_25 AT %MX26508.25 : BOOL;
	bArm2VertStn2Down_26 AT %MX26508.26 : BOOL;
	bArm2VertStn2Down_27 AT %MX26508.27 : BOOL;
	bArm2VertStn2Down_28 AT %MX26508.28 : BOOL;
	bArm2VertStn2Down_29 AT %MX26508.29 : BOOL;
	bArm2VertStn2Down_30 AT %MX26508.30 : BOOL;
	bArm2VertStn2Down_31 AT %MX26508.31 : BOOL;

	bArm2VertStn3Down_00 AT %MX26512.0 : BOOL;
	bArm2VertStn3Down_01 AT %MX26512.1 : BOOL;
	bArm2VertStn3Down_02 AT %MX26512.2 : BOOL;
	bArm2VertStn3Down_03 AT %MX26512.3 : BOOL;
	bArm2VertStn3Down_04 AT %MX26512.4 : BOOL;
	bArm2VertStn3Down_05 AT %MX26512.5 : BOOL;
	bArm2VertStn3Down_06 AT %MX26512.6 : BOOL;
	bArm2VertStn3Down_07 AT %MX26512.7 : BOOL;
	bArm2VertStn3Down_08 AT %MX26512.8 : BOOL;
	bArm2VertStn3Down_09 AT %MX26512.9 : BOOL;
	bArm2VertStn3Down_10 AT %MX26512.10 : BOOL;
	bArm2VertStn3Down_11 AT %MX26512.11 : BOOL;
	bArm2VertStn3Down_12 AT %MX26512.12 : BOOL;
	bArm2VertStn3Down_13 AT %MX26512.13 : BOOL;
	bArm2VertStn3Down_14 AT %MX26512.14 : BOOL;
	bArm2VertStn3Down_15 AT %MX26512.15 : BOOL;
	bArm2VertStn3Down_16 AT %MX26512.16 : BOOL;
	bArm2VertStn3Down_17 AT %MX26512.17 : BOOL;
	bArm2VertStn3Down_18 AT %MX26512.18 : BOOL;
	bArm2VertStn3Down_19 AT %MX26512.19 : BOOL;
	bArm2VertStn3Down_20 AT %MX26512.20 : BOOL;
	bArm2VertStn3Down_21 AT %MX26512.21 : BOOL;
	bArm2VertStn3Down_22 AT %MX26512.22 : BOOL;
	bArm2VertStn3Down_23 AT %MX26512.23 : BOOL;
	bArm2VertStn3Down_24 AT %MX26512.24 : BOOL;
	bArm2VertStn3Down_25 AT %MX26512.25 : BOOL;
	bArm2VertStn3Down_26 AT %MX26512.26 : BOOL;
	bArm2VertStn3Down_27 AT %MX26512.27 : BOOL;
	bArm2VertStn3Down_28 AT %MX26512.28 : BOOL;
	bArm2VertStn3Down_29 AT %MX26512.29 : BOOL;
	bArm2VertStn3Down_30 AT %MX26512.30 : BOOL;
	bArm2VertStn3Down_31 AT %MX26512.31 : BOOL;

